FUNCTION "FC21 Ventil 1A0-2E" : VOID	// FC 21
TITLE = Block for valve actuation and fault monitoring
//Erstellung:
//Datum        Bearbeiter                                                 Version
//--------------------------------------------------------------------------------
//26.06.97     H.Rüttling (rh)                                            01.00.00
//
//Änderungen:
//Nr. Datum    Bearb Änderung                                       Marke  Version
//--------------------------------------------------------------------------------
//01  09.02.99 sra   Einfügen der Handbedienuung                    ()    01.01.00
//02  16.04.99 sra   Fehlerbeseitigung Störungsquittierung          ()    01.01.01
//03  21.05.99 jm    Ventiltyp 0 eingefügt                          ()    01.02.00
//04  23.07.99 sra   Ausg. wird auch bei Simulation gesetzt         ()    01.02.01
//06  18.09.00 sra   komplette Überarbeitung / neue Struktur        ()    02.00.00
//07  31.10.05 sra   Ansteuerung Handbedienung im Automode rücksetz.
//                   Handbedienung zentral sperren                  (007) 02.01.00
//08  04.09.06 sra   Änderung Störungsquittierung                   (008) 02.02.00
//09  18.02.09 kmj   Objektststatus für OP ergänzt                  (009) 02.03.00
//10  20.03.09 kal   Objektststatus für OP ergänzt (überarbeitet)   (010) 02.03.01
//11  25.03.09 kal   1A0E-Objekt kann verzögert "in Betrieb" melden (011) 02.03.02
//12  25.03.09 kal   INC nach + geändert                            (012) 02.03.03
//13  20.11.07 gea   Handmode zurücksetzen wenn Handmode gesperrt   (013) 02.03.04
//14  14.07.09 kal   Objektstatus überarbeitet                      (014) 02.03.05
//15  05.12.13 sra   "Anlage ein" eingefügt (Not-Aus-Konzept)       (015) 02.04.00
//________________________________________________________________________________
//Funktion:
//
//-Der Parameter VENTIL_TYP unterscheidet zwischen 4 verschiedenen Ventiltypen
// Typ 0 = Ventil ohne Rückmeldung
// Typ 1 = Ventil oder Klappe mit der Rückmeldung angesteuert und nicht 
//        angesteuert: 1. Ausgang auf, Eingang auf, Eingang zu
//                     2. Ausgang zu , Eingang zu , Eingang auf
// TYP 2 = Ventil oder Klappe mit der Rückmeldung angesteuert
//                     1. Ausgang auf, Eingang auf
//                     2. Ausgang zu , Eingang zu 
// TYP 3 = Ventil oder Klappe mit der Rückmeldung nicht angesteuert
//                     1. Ausgang auf, Eingang zu
//                     2. Ausgang zu , Eingang auf 
//
//-Der Baustein steuert den Ablauf eines Ventils mit 1 Ausgang und 0-2 Eingängen
// durch setzten des Eingangsparameters "in_Ansteuerung_Ventil".
//
//-Der Ausgang wird nur angesteuert wenn der Eingang "in_Anlage_ein" = true
// ist. Diese Funktion ist vorhanden, um bei einem Not-Halt die Anlage vor 
// unkontrolliertem Einschalten zu schützen. 
//
//-Ist in der Ventilstruktur die Taktfunktion freigegeben wird bei Freigabe des 
// Ventils der Ausgang entsprechend der Impuls-/Pausezeit angesteuert.
//
//-Der Baustein überwacht den Zustand des Ausgangs und der Eingänge und generiert 
// nach Ablauf der "Sollzeit Störung" eine Störmeldung
//
//-Ist das Bit "Simulation" auf TRUE, so werden die Eingänge simuliert.
//
//-Ist die Kennung "Schalthäufigkeitszähler_ein" aktiviert werden die
// Ansteuerungen des Ventils aufsummiert. Dies erfolgt mit setzen des Ausgangs.
//
//-Der Baustein kopiert die Parameter "in_Eingang_...", "io_Ausgang_Ventil", 
// "in_Quitt_Stoerung" und "io_Stoerung" in die angegebene Datenstruktur zur 
// Visualisierung auf einem Farbgrafiksystem. Diese Parameter müssen folglich 
// nicht mehr extern umkopiert werden.
//
//-Ist der Parameter "in_Handbedienung_erlaubt" angewählt kann das Ventil über 
// eine Farbgrafik oder ein Bedienterminal manuell angesteuert werden
//
AUTHOR : rh
FAMILY : AZO
VERSION : 0.0
VAR_INPUT
  in_Ventil_Typ : INT ;	//see Functional description below
  in_Handbedienung_erlaubt : BOOL ;	//1 = manual operation permitted, 0 = manual operation not permitted/locked
  in_Quitt_Stoerung_noetig : BOOL ;	//1 = fault acknowledgement required, 0 = automatic fault acknowledgement
  in_Quitt_Stoerung : BOOL ;	//Fault acknowledgement when fault_acknowledgement_required = 1
  in_Anlage_ein : BOOL ;	//Anlage bzw. Anlagenbereich nach Not-Halt freigegeben
  in_Ansteuerung_Ventil : BOOL ;	//Actuation of valve in automatic mode
  in_Eingang_angesteuert : BOOL ;	//Valve intake when actuated
  in_Eingang_nicht_angest : BOOL ;	//Valve intake when not actuated
END_VAR
VAR_IN_OUT
  io_Ausgang_Ventil : BOOL ;	//Valve outlet
  io_Ventil_in_Betrieb : BOOL ;	//Signal "valve in operation" (actuated)
  io_Stoerung : BOOL ;	//Signal "valve fault"
  io_Ventilstruktur : ANY ;	//ANY pointer of valve structure
END_VAR
VAR_TEMP
  Freigabe_Takt : BOOL ;
  Rueckmeldung : BOOL ;
  Start_mit_Impuls : BOOL ;
  Dauertakt : BOOL ;
  Taktausgang : BOOL ;
  Taktanzahl_erreicht : BOOL ;
  Diskrepanz : BOOL ;
  positive_Flanke : BOOL ;
  Impulszeit : REAL ;
  Pausezeit : REAL ;
  Sollanzahl_Takte : INT ;
  Zeitzaehler : REAL ;
  Taktzaehler : INT ;
  Objektstatus : INT ;
END_VAR
BEGIN
NETWORK
TITLE = Anfangs-DW der Struktur aus ANY-Zeiger auslesen
      L     P##io_Ventilstruktur;
      LAR2;
      L     D [AR2,P#6.0];
      LAR2;
NETWORK
TITLE = Simulation
      AN    DIX [AR2,P#3.5];	// Simulation ein (Struktur)
      JC    ESIM;
      A     #io_Ausgang_Ventil;
      =     #in_Eingang_angesteuert;
      AN    #io_Ausgang_Ventil;
      =     #in_Eingang_nicht_angest;
      L     #in_Ventil_Typ;
      L     3;
      <>I;
      JC    ESIM;
      CLR;
      =     #in_Eingang_angesteuert;
      AN    #io_Ausgang_Ventil;
      =     #in_Eingang_nicht_angest;
ESIM: NOP   0;
NETWORK
TITLE = Umschaltung Hand-/Automatikmode 
      A     DIX [AR2,P#2.7];	// Handmode von Farbgrafik (Struktur)
      AN    DIX [AR2,P#3.1];	// Handmode gesperrt (Struktur)
      AN    "M0.0 LockManualMode";	// Handbedienung zentral sperren (007)
      S     DIX [AR2,P#2.6];	// Handmode zu Farbgrafik (Struktur)
      ON    DIX [AR2,P#2.7];	// Handmode von Farbgrafik (Struktur)
      ON    #in_Handbedienung_erlaubt;
      O     "M0.0 LockManualMode";	// Handbedienung zentral sperren (007)
      O     DIX [AR2,P#3.1];	// Handmode gesperrt (Struktur)//(013)
      R     DIX [AR2,P#2.6];	// Handmode zu Farbgrafik (Struktur)
      R     DIX [AR2,P#2.7];	// Handmode von Farbgrafik (Struktur) (007)
NETWORK
TITLE = Ansteuerung Handmode zurücksetzen
//(007) 
      AN    DIX [AR2,P#2.6];	// Handmode zu Farbgrafik (Struktur)
      R     DIX [AR2,P#3.0];	// Ansteuerung Handmode von Farbgrafik (Struktur)
NETWORK
TITLE = Daten für Takt in temporäre Variablen laden
      A     #in_Anlage_ein;	// (015)
      A     #in_Ansteuerung_Ventil;
      A     DIX [AR2,P#3.6];	// Freigabe Takt (Struktur)
      =     #Freigabe_Takt;
      A     DIX [AR2,P#3.2];	// Start mit Impuls (Struktur)
      =     #Start_mit_Impuls;
      A     DIX [AR2,P#3.3];	// Taktanzahl erreicht (Struktur)
      =     #Taktanzahl_erreicht;
      A     DIX [AR2,P#3.4];	// Dauertakt (Struktur)
      =     #Dauertakt;
      A     DIX [AR2,P#3.7];	// Taktausgang (Struktur)
      =     #Taktausgang;
      L     DID [AR2,P#8.0];	// Impulszeit (Struktur)
      T     #Impulszeit;
      L     DID [AR2,P#12.0];	// Pausezeit (Struktur)
      T     #Pausezeit;
      L     DID [AR2,P#16.0];	// Impuls-/Pausezähler (Struktur)
      T     #Zeitzaehler;
      L     DIW [AR2,P#20.0];	// Sollanzahl Takte (Struktur)
      T     #Sollanzahl_Takte;
      L     DIW [AR2,P#22.0];	// Taktzähler (Struktur)
      T     #Taktzaehler;
NETWORK
TITLE = Rückmeldung für Takt
      A(;
      L     #in_Ventil_Typ;
      L     0;
      ==I;
      );
      A     #io_Ausgang_Ventil;
      O;
      A(;
      L     #in_Ventil_Typ;
      L     1;
      ==I;
      );
      A     #in_Eingang_angesteuert;
      O;
      A(;
      L     #in_Ventil_Typ;
      L     2;
      ==I;
      );
      A     #in_Eingang_angesteuert;
      O;
      A(;
      L     #in_Ventil_Typ;
      L     3;
      ==I;
      );
      AN    #in_Eingang_nicht_angest;
      =     #Rueckmeldung;
NETWORK
TITLE = Takt generieren
      CALL  "FC2 Taktgeber_Timernachb" (
           in_Freigabe              := #Freigabe_Takt,
           in_Rueckmeldung          := #Rueckmeldung,
           in_Start_mit_Impuls      := #Start_mit_Impuls,
           in_Dauertakt             := #Dauertakt,
           in_Impuls                := "M1.7 ClockTimerFunction",
           in_Impulszeit_in_100ms   := "MW 6 Timer Val Cycle FCs",
           in_Impulszeit            := #Impulszeit,
           in_Pausezeit             := #Pausezeit,
           in_Sollanzahl_Takte      := #Sollanzahl_Takte,
           io_Taktausgang           := #Taktausgang,
           io_Taktanzahl_erreicht   := #Taktanzahl_erreicht,
           io_Zeitzaehler           := #Zeitzaehler,
           io_Taktzaehler           := #Taktzaehler);
NETWORK
TITLE = Ansteuerung Ventil
      A     #in_Anlage_ein;	// (015)
      A(;
      ON    #in_Quitt_Stoerung_noetig;
      O;
      A     #in_Quitt_Stoerung_noetig;
      AN    #io_Stoerung;
      );
      A(;
      AN    DIX [AR2,P#2.6];	// Automatikmode zu Farbgrafik (Struktur)
      AN    DIX [AR2,P#3.6];	// Freigabe Takt (Struktur)
      A     #in_Ansteuerung_Ventil;
      O;
      AN    DIX [AR2,P#2.6];	// Automatikmode zu Farbgrafik (Struktur)
      A     DIX [AR2,P#3.6];	// Freigabe Takt (Struktur)
      A     #Taktausgang;
      O;
      A     DIX [AR2,P#2.6];	// Handmode zu Farbgrafik (Struktur)
      A     DIX [AR2,P#3.0];	// Ansteuerung Handmode von Farbgrafik (Struktur)
      );
      =     #io_Ausgang_Ventil;
NETWORK
TITLE = Ventiltyp festlegen
      L     #in_Ventil_Typ;
      L     0;
      ==I;
      JC    TYP0;	// Sprung zu Ventil Typ 0
      TAK;
      L     1;
      ==I;
      JC    TYP1;	// Sprung zu Ventil Typ 1
      TAK;
      L     2;
      ==I;
      JC    TYP2;	// Sprung zu Ventil Typ 2
      TAK;
      L     3;
      ==I;
      JC    TYP3;	// Sprung zu Ventil Typ 3
      JU    ENDE;
NETWORK
TITLE = Betriebsmeldung Typ 0 (kein Eingang)
TYP0: A     #io_Ausgang_Ventil;
      A(;	// (011)
      L     DIW [AR2,P#40.0];	// (011) Istzeit Verzögerung (Struktur) 
      L     DIW [AR2,P#38.0];	// (011) Sollzeit Verzögerung (Struktur)
      >=I;	// (011)
      );	// (011)
      =     #io_Ventil_in_Betrieb;	// Betriebsmeldung anzeigen
NETWORK
TITLE = Istzähler Verzögerung hochzählen (011)
      A     #io_Ausgang_Ventil;
      AN    "M4.5 ImpulseClock1,0Sec";	// Sekundenimpuls (Standardmerker)
      O     #io_Ventil_in_Betrieb;	// Betriebsmeldung anzeigen
      JC    KVZ;
      L     DIW [AR2,P#40.0];	// Istzeit Verzögerung (Struktur)
      +     1;
      T     DIW [AR2,P#40.0];	// Istzeit Verzögerung (Struktur)
KVZ:  NOP   0;
NETWORK
TITLE = Istzähler Verzögerung zurücksetzen (011)
      O     #io_Ausgang_Ventil;
      JC    RVZ;
      L     0;
      T     DIW [AR2,P#40.0];	// Istzeit Verzögerung (Struktur)
RVZ:  NOP   0;
NETWORK
TITLE = Diskrepanz Typ 0 (kein Eingang)
      CLR;	// keine Diskrepanz möglich
      =     #Diskrepanz;
      JU    STOE;
NETWORK
TITLE = Betriebsmeldung Typ1 (Eingang angesteuert und nicht angesteuert)
TYP1: A     #io_Ausgang_Ventil;
      A     #in_Eingang_angesteuert;
      AN    #in_Eingang_nicht_angest;
      =     #io_Ventil_in_Betrieb;
NETWORK
TITLE = Diskrepanz Typ 1 (Eingang angesteuert und nicht angesteuert)
      A     #io_Ausgang_Ventil;
      AN    #in_Eingang_angesteuert;
      O;
      AN    #io_Ausgang_Ventil;
      AN    #in_Eingang_nicht_angest;
      O;
      A     #in_Eingang_angesteuert;
      A     #in_Eingang_nicht_angest;
      O;
      AN    #in_Eingang_angesteuert;
      AN    #in_Eingang_nicht_angest;
      =     #Diskrepanz;
      JU    STOE;
NETWORK
TITLE = Betriebsmeldung Typ 2 (Eingang angesteuert)
TYP2: A     #io_Ausgang_Ventil;
      A     #in_Eingang_angesteuert;
      =     #io_Ventil_in_Betrieb;
NETWORK
TITLE = Diskrepanz Typ 2 (Eingang angesteuert)
      A     #io_Ausgang_Ventil;
      AN    #in_Eingang_angesteuert;
      O;
      AN    #io_Ausgang_Ventil;
      A     #in_Eingang_angesteuert;
      =     #Diskrepanz;
      JU    STOE;
NETWORK
TITLE = Betriebsmeldung Typ 3 (Eingang nicht angesteuert)
TYP3: A     #io_Ausgang_Ventil;
      AN    #in_Eingang_nicht_angest;
      =     #io_Ventil_in_Betrieb;
NETWORK
TITLE = Diskrepanz Typ 3 (Eingang nicht angesteuert)
      A     #io_Ausgang_Ventil;
      A     #in_Eingang_nicht_angest;
      O;
      AN    #io_Ausgang_Ventil;
      AN    #in_Eingang_nicht_angest;
      =     #Diskrepanz;
NETWORK
TITLE = Störungszähler
STOE: A     #in_Quitt_Stoerung_noetig;
      AN    #in_Quitt_Stoerung;
      A     #io_Stoerung;
      O;
      A     #Diskrepanz;
      AN    #in_Quitt_Stoerung;	// (008)
      O;	// (008)
      AN    #in_Quitt_Stoerung_noetig;	// (008)
      A     #Diskrepanz;	// (008)
      JC    SZ1;
      L     0;	// Wenn keine Diskrepanz dann Zähler löschen
      T     DIW [AR2,P#6.0];	// Istzeit Störung (Struktur)
      JU    ESZ;
// Störungszähler in jeder Sekunde erhöhen
SZ1:  O     #io_Stoerung;
      ON    "M4.5 ImpulseClock1,0Sec";	// Sekundenimpuls (Standardmerker)
      JC    ESZ;
      L     DIW [AR2,P#6.0];	// Istzeit Störung (Struktur)
      +     1;	// (012)
      T     DIW [AR2,P#6.0];	// Istzeit Störung (Struktur)
ESZ:  NOP   0;
NETWORK
TITLE = Störmeldung ausgeben
      L     DIW [AR2,P#6.0];	// Istzeit Störung (Struktur)
      L     DIW [AR2,P#4.0];	// Sollzeit Störung (Struktur)
      >=I;
      =     #io_Stoerung;
NETWORK
TITLE = Stoerung quittieren
      O     #Diskrepanz;	// Stoerung steht noch an
      ON    #io_Stoerung;
      JC    ESQ;
      ON    #in_Quitt_Stoerung_noetig;	// Stoerung muß quittiert werden ?
      JC    SQ1;	// Stoerung muß nicht quittiert werden
      A     #in_Quitt_Stoerung;
SQ1:  R     #io_Stoerung;
ESQ:  NOP   0;
NETWORK
TITLE = Flankenauswertung Ausgang Ventil für Schalthäufigkeitzähler
      A     #io_Ausgang_Ventil;
      FP    DIX [AR2,P#24.3];	// Flankenmerker Ausgang (Struktur)
      =     #positive_Flanke;
NETWORK
TITLE = Schalthäufigkeitzähler
      ON    DIX [AR2,P#0.3];	// Kennung Schalthäufigkeitzähler ein (Struktur)
      ON    #positive_Flanke;
      JC    ESHZ;
      L     1.000000e+00;
      L     DID [AR2,P#26.0];	// Schalthäufigkeitzähler (Struktur)
      +R;
      T     DID [AR2,P#26.0];	// Schalthäufigkeitzähler (Struktur)
ESHZ: NOP   0;
NETWORK
TITLE = Schalthäufigkeitzähler zurücksetzten
      AN    DIX [AR2,P#24.0];	// Reset Schalthäufigkeitzähler (Struktur)
      JC    E_RS;
      L     0.000000e+00;
      T     DID [AR2,P#26.0];	// Schalthäufigkeitzähler (Struktur)
      CLR;
      =     DIX [AR2,P#24.0];	// Reset Schalthäufigkeitzähler (Struktur)
E_RS: NOP   0;
NETWORK
TITLE = Warnmeldung Schalthäufigkeitszähler erzeugen
      A(;
      L     DID [AR2,P#26.0];	// Schalthäufigkeitzähler (Struktur)
      L     DID [AR2,P#30.0];	// Sollwert Warnung (Struktur)
      >R;
      );
      A(;
      L     DID [AR2,P#30.0];	// Sollwert Warnung (Struktur)
      L     0.000000e+00;
      <>R;
      );
      =     DIX [AR2,P#24.1];	// Warnmeldung Schalthäufigkeitzähler (Struktur)
NETWORK
TITLE = Alarmmeldung Schalthäufigkeitszähler erzeugen
      A(;
      L     DID [AR2,P#26.0];	// Schalthäufigkeitzähler (Struktur)
      L     DID [AR2,P#34.0];	// Sollwert Alarm (Struktur)
      >R;
      );
      A(;
      L     DID [AR2,P#34.0];	// Sollwert Alarm (Struktur)
      L     0.000000e+00;
      <>R;
      );
      =     DIX [AR2,P#24.2];	// Alarmmeldung Schalthäufigkeitzähler (Struktur)
NETWORK
TITLE =  Objektstatus für Visualisation OP (009) (010)
//Stati:
//-------
//1 = nicht in Betrieb, keine Störung ==> Farbvorschlag weiß
//5 = angesteuert, in Betrieb, keine Störung ==> Farbvorschlag grün
//9 = angesteuert, nicht in Betrieb, keine Störung ==> Farbvorschlag grau
//16 = Störung ==> Farbvorschlag rot
// 1 = nicht in Betrieb, keine Störung ==> Farbvorschlag weiß
      L     1;
      AN    #io_Ausgang_Ventil;
      AN    #io_Stoerung;
      AN    DIX [AR2,P#1.3];	// (014) Kennung "invers"
      O;
      A     #io_Ausgang_Ventil;
      A     #io_Ventil_in_Betrieb;
      AN    #io_Stoerung;
      A     DIX [AR2,P#1.3];	// (014) Kennung "invers"
      JC    disp;
// 5 = angesteuert, in Betrieb, keine Störung ==> Farbvorschlag grün
      L     5;
      A     #io_Ausgang_Ventil;
      A     #io_Ventil_in_Betrieb;
      AN    #io_Stoerung;
      AN    DIX [AR2,P#1.3];	// (014) Kennung "invers"
      O;
      AN    #io_Ausgang_Ventil;
      AN    #io_Stoerung;
      A     DIX [AR2,P#1.3];	// (014) Kennung "invers"
      JC    disp;
// 9 = angesteuert, nicht in Betrieb, keine Störung ==> Farbvorschlag grau
      L     9;
      A     #io_Ausgang_Ventil;
      AN    #io_Ventil_in_Betrieb;
      AN    #io_Stoerung;
      JC    disp;
// 16 = Störung ==> Farbvorschlag rot
      L     16;
      A     #io_Stoerung;
      JC    disp;
      L     0;
disp: T     #Objektstatus;
NETWORK
TITLE = Daten in Struktur speichern
      A     #in_Anlage_ein;	// (015)
      =     DIX [AR2,P#42.0];	// (015) Anlage ein (Struktur)
      A     #in_Eingang_angesteuert;
      =     DIX [AR2,P#2.1];	// Eingang angesteuert (Struktur)
      A     #in_Eingang_nicht_angest;
      =     DIX [AR2,P#2.2];	// Eingang nicht angesteuert (Struktur)
      A     #io_Ausgang_Ventil;
      =     DIX [AR2,P#2.0];	// Ausgang Ventil (Struktur)
      A     #io_Ventil_in_Betrieb;
      =     DIX [AR2,P#2.4];	// Ventil in Betrieb (Struktur)
      A     #io_Stoerung;
      =     DIX [AR2,P#2.5];	// Störung (Struktur)
      A     #Taktanzahl_erreicht;
      =     DIX [AR2,P#3.3];	// Taktanzahl erreicht (Struktur)
      A     #Taktausgang;
      =     DIX [AR2,P#3.7];	// Taktausgang (Struktur)
      L     #Zeitzaehler;
      T     DID [AR2,P#16.0];	// Impuls-/Pausezähler (Struktur)
      L     #Taktzaehler;
      T     DIW [AR2,P#22.0];	// Taktzähler (Struktur)
      L     #Objektstatus;	// (009)
      T     DIW [AR2,P#48.0];	// #Objektstatus  (Struktur)   // (009)
NETWORK
TITLE = ENDE
ENDE: NOP   0;
END_FUNCTION

FUNCTION "FC22 Ventil 2A2E" : VOID	// FC 22
TITLE = Block for valve actuation and fault monitoring 2O,2I
//Erstellung:
//Datum        Bearbeiter                                                 Version
//--------------------------------------------------------------------------------
//24.09.98     A.Geiger (gea)                                             01.00.00
//
//Änderungen:
//Nr. Datum    Bearb Änderung                                       Marke  Version
//--------------------------------------------------------------------------------
//01  16.04.99 sra   Fehlerbeseitigung Störungsquittierung          ()    01.00.01
//02  21.05.99 sra   Einfügen der Handbedienuung                    ()    01.01.00
//03  23.07.99 sra   Ausg. wird auch bei Simulation gesetzt         ()    01.01.01
//04  19.10.99 sra   Anpassung an neue Struktur                     ()    01.02.00
//05  19.09.00 sra   komplette Überarbeitung / neue Struktur        ()    02.00.00
//06  15.02.01 sra   Rücksetzen Istwert Störung bei Quitt.          ()    02.00.01
//07  31.03.03 sra   Fehlerbeseitigung Störungsquittierung          (007) 02.00.02
//08  23.03.05 sra   Änderung Störungsquittierung                   (008) 02.01.00
//09  31.10.05 sra   Ansteuerung Handbedienung im Automode rücksetz.
//                   Handbedienung zentral sperren                  (009) 02.02.00
//10  03.05.06 gea   Fehlerbeseitigung Störungszähler               (010) 02.02.01
//11  18.02.09 kmj   Objektstatus ergänzt                           (011) 02.03.00
//12  20.03.09 kal   Objektstatus ergänzt (überarbeitet)            (012) 02.03.01
//13  24.04.09 gea   Handmode zurücksetzen wenn Handmode gesperrt   (013) 02.03.02
//14  10.09.09 sra   Objektststatus für OP ergänzt (erweitert)      (014) 02.04.00
//15  15.10.09 gea   Korrektur Taktpause                            (015) 02.04.01
//16  26.03.12 jm    Objektstatus korrigiert                        (016) 02.04.02
//17  07.09.12 jm    Ohjektstatus aufgeteilt (3 Versionen)          (017) 02.04.03
//18  12.10.12 jm    Objektstatus 3 optimiert                       (018) 02.04.04
//19  15.10.12 jm    Objektstatus 3 optimiert (1,6 anstatt 1,5)     (019) 02.04.05
//20  18.12.12 sra   Kennung links rechts eingefügt                 (020) 02.05.00
//21  05.12.13 sra   "Anlage ein" eingefügt (Not-Aus-Konzept)       (021) 02.06.00
//22  24.07.14 jm    Ohjektstatus ergänzt/geändert                  (022) 02.07.01
//23  09.03.16 jm    Objektstatus 9/19 bis Ende oder Störung        (023) 02.07.02
//________________________________________________________________________________
//Funktion:
//
//-Der Baustein steuert den Ablauf eines Ventils mit 2 Ausgängen und 2 Eingängen.
//
//-Die Ausgänge werden nur angesteuert wenn der Eingang "in_Anlage_ein" = true
// ist. Diese Funktion ist vorhanden, um bei einem Not-Halt die Anlage vor 
// unkontrolliertem Einschalten zu schützen. 
//
//-Ist in der Ventilstruktur die Taktfunktion freigegeben wird bei Freigabe des 
// Ventils der Ausgang entsprechend der Impuls-/Pausezeit angesteuert.
//
//-Der Baustein überwacht den Zustand der Ausgänge und der Eingänge und generiert 
// nach Ablauf der "Sollzeit Störung" eine Störmeldung
//
//-Ist das Bit "Simulation" auf TRUE, so werden die Eingänge simuliert.
//
//-Ist die Kennung "Schalthäufigkeitszähler_ein" aktiviert werden die
// Ansteuerungen des Ventils aufsummiert. Dies erfolgt mit setzen des Ausgangs.
//
//-Der Baustein kopiert die Parameter "in_Eingang_...", "io_Ausgang_...", 
// "in_Quitt_Stoerung" und "io_Stoerung" in die angegebene Datenstruktur zur 
// Visualisierung auf einem Farbgrafiksystem. Diese Parameter müssen folglich 
// nicht mehr extern umkopiert werden.
//
//-Ist der Parameter "in_Handbedienung_erlaubt" angewählt kann das Ventil über 
// eine Farbgrafik oder ein Bedienterminal manuell angesteuert werden
//
AUTHOR : gea
FAMILY : AZO
NAME : standard
VERSION : 0.0
VAR_INPUT
  in_Handbedienung_erlaubt : BOOL ;	//1 = manual operation permitted, 0 = manual operation not permitted/locked
  in_Quitt_Stoerung_noetig : BOOL ;	//1 = fault acknowledgement required, 0 = automatic fault acknowledgement
  in_Quitt_Stoerung : BOOL ;	//Fault acknowledgement when fault_acknowledgement_required = 1
  in_Anlage_ein : BOOL ;	//Anlage bzw. Anlagenbereich nach Not-Halt freigegeben
  in_Ansteuerung_Stellung1 : BOOL ;	//Actuation of valve position 1 in automatic mode
  in_Ansteuerung_Stellung2 : BOOL ;	//Actuation of valve position 2 in automatic mode
  in_Eingang_Stellung_1 : BOOL ;	//Valve intake when position 1 actuated
  in_Eingang_Stellung_2 : BOOL ;	//Valve intake when position 2 actuated
END_VAR
VAR_IN_OUT
  io_Ausgang_Stellung_1 : BOOL ;	//Valve output to actuate position 1
  io_Ausgang_Stellung_2 : BOOL ;	//Valve output to actuate position 2
  io_Stellung_1_Betrieb : BOOL ;	//Signal "position 1 in operation" (position 1 actuated)
  io_Stellung_2_Betrieb : BOOL ;	//Signal "position 2 in operation" (position 2 actuated)
  io_Stoerung : BOOL ;	//Signal "valve fault"
  io_Ventilstruktur : ANY ;	//ANY pointer of valve structure
END_VAR
VAR_TEMP
  Freigabe_Takt : BOOL ;
  Rueckmeldung : BOOL ;
  Start_mit_Impuls : BOOL ;
  Dauertakt : BOOL ;
  Taktausgang : BOOL ;
  Taktanzahl_erreicht : BOOL ;
  Diskrepanz : BOOL ;
  positive_Flanke : BOOL ;
  Impulszeit : REAL ;
  Pausezeit : REAL ;
  Sollanzahl_Takte : INT ;
  Zeitzaehler : REAL ;
  Taktzaehler : INT ;
  Objektstatus : INT ;
END_VAR
BEGIN
NETWORK
TITLE = Anfangs-DW der Struktur aus ANY-Zeiger auslesen
      L     P##io_Ventilstruktur;
      LAR2;
      L     D [AR2,P#6.0];
      LAR2;
NETWORK
TITLE = Simulation
      AN    DIX [AR2,P#4.1];	// Simulation ein (Struktur)
      JC    ESIM;
      A     #io_Ausgang_Stellung_1;
      AN    #io_Ausgang_Stellung_2;
      O;
      AN    #io_Ausgang_Stellung_2;
      AN    DIX [AR2,P#2.2];	// Eingang Stellung 1 (Struktur)
      AN    DIX [AR2,P#2.3];	// Eingang Stellung 2 (Struktur)
      O;
      AN    #io_Ausgang_Stellung_1;
      AN    #io_Ausgang_Stellung_2;
      A     DIX [AR2,P#2.2];	// Eingang Stellung 1 (Struktur)
      S     #in_Eingang_Stellung_1;
      R     #in_Eingang_Stellung_2;
      AN    #io_Ausgang_Stellung_1;
      A     #io_Ausgang_Stellung_2;
      O;
      AN    #io_Ausgang_Stellung_1;
      AN    #io_Ausgang_Stellung_2;
      A     DIX [AR2,P#2.3];	// Eingang Stellung 2 (Struktur)
      R     #in_Eingang_Stellung_1;
      S     #in_Eingang_Stellung_2;
ESIM: NOP   0;
NETWORK
TITLE = Umschaltung Hand-/Automatikmode 
      A     DIX [AR2,P#3.2];	// Handmode von Farbgrafik (Struktur)
      AN    DIX [AR2,P#3.5];	// Handmode gesperrt (Struktur)
      AN    "M0.0 LockManualMode";	// Handbedienung zentral sperren (009)
      S     DIX [AR2,P#3.1];	// Handmode zu Farbgrafik (Struktur)
      ON    DIX [AR2,P#3.2];	// Handmode von Farbgrafik (Struktur)
      ON    #in_Handbedienung_erlaubt;
      O     "M0.0 LockManualMode";	// Handbedienung zentral sperren (009)
      O     DIX [AR2,P#3.5];	// Handmode gesperrt (Struktur) (013)
      R     DIX [AR2,P#3.1];	// Handmode zu Farbgrafik (Struktur)
      R     DIX [AR2,P#3.2];	// Handmode von Farbgrafik (Struktur) (009)
NETWORK
TITLE = Ansteuerung Handmode zurücksetzen
//(009) 
      AN    DIX [AR2,P#3.1];	// Handmode zu Farbgrafik (Struktur)
      R     DIX [AR2,P#3.3];	// Ansteuerung Stellung 1 Handmode von Farbgrafik (Struktur)
      R     DIX [AR2,P#3.4];	// Ansteuerung Stellung 2 Handmode von Farbgrafik (Struktur)
NETWORK
TITLE = Daten für Takt in temporäre Variablen laden
      A     #in_Anlage_ein;	// (021)
      A(;
      O     #in_Ansteuerung_Stellung1;
      O     #in_Ansteuerung_Stellung2;
      );
      A     DIX [AR2,P#4.2];	// Freigabe Takt (Struktur)
      =     #Freigabe_Takt;
      A     DIX [AR2,P#3.6];	// Start mit Impuls (Struktur)
      =     #Start_mit_Impuls;
      A     DIX [AR2,P#3.7];	// Taktanzahl erreicht (Struktur)
      =     #Taktanzahl_erreicht;
      A     DIX [AR2,P#4.0];	// Dauertakt (Struktur)
      =     #Dauertakt;
      A     DIX [AR2,P#4.3];	// Taktausgang (Struktur)
      =     #Taktausgang;
      L     DID [AR2,P#10.0];	// Impulszeit (Struktur)
      T     #Impulszeit;
      L     DID [AR2,P#14.0];	// Pausezeit (Struktur)
      T     #Pausezeit;
      L     DID [AR2,P#18.0];	// Impuls-/Pausezähler (Struktur)
      T     #Zeitzaehler;
      L     DIW [AR2,P#22.0];	// Sollanzahl Takte (Struktur)
      T     #Sollanzahl_Takte;
      L     DIW [AR2,P#24.0];	// Taktzähler (Struktur)
      T     #Taktzaehler;
NETWORK
TITLE = Rückmeldung für Takt
// (network holds code this reader does not know; not shown)
NETWORK
TITLE = Takt generieren
      CALL  "FC2 Taktgeber_Timernachb" (
           in_Freigabe              := #Freigabe_Takt,
           in_Rueckmeldung          := #Rueckmeldung,
           in_Start_mit_Impuls      := #Start_mit_Impuls,
           in_Dauertakt             := #Dauertakt,
           in_Impuls                := "M1.7 ClockTimerFunction",
           in_Impulszeit_in_100ms   := "MW 6 Timer Val Cycle FCs",
           in_Impulszeit            := #Impulszeit,
           in_Pausezeit             := #Pausezeit,
           in_Sollanzahl_Takte      := #Sollanzahl_Takte,
           io_Taktausgang           := #Taktausgang,
           io_Taktanzahl_erreicht   := #Taktanzahl_erreicht,
           io_Zeitzaehler           := #Zeitzaehler,
           io_Taktzaehler           := #Taktzaehler);
NETWORK
TITLE = Ansteuerung Stellung 1
      A     #in_Anlage_ein;	// (021)
      A(;
      ON    #in_Quitt_Stoerung_noetig;
      O;
      A     #in_Quitt_Stoerung_noetig;
      AN    #io_Stoerung;
      );
      A(;
      AN    DIX [AR2,P#3.1];	// Automatikmode zu Farbgrafik (Struktur)
      AN    DIX [AR2,P#4.2];	// Freigabe Takt (Struktur)
      A     #in_Ansteuerung_Stellung1;
      AN    #in_Ansteuerung_Stellung2;
      O;
      AN    DIX [AR2,P#3.1];	// Automatikmode zu Farbgrafik (Struktur)
      A     DIX [AR2,P#4.2];	// Freigabe Takt (Struktur)
      A     #Taktausgang;
      O;
      A     DIX [AR2,P#3.1];	// Handmode zu Farbgrafik (Struktur)
      A     DIX [AR2,P#3.3];	// Ansteuerung Stellung 1 Handmode von Farbgrafik (Struktur)
      AN    DIX [AR2,P#3.4];	// Ansteuerung Stellung 2 Handmode von Farbgrafik (Struktur)
      );
      =     #io_Ausgang_Stellung_1;
NETWORK
TITLE = Ansteuerung Stellung 2
      A     #in_Anlage_ein;	// (021)
      A(;
      ON    #in_Quitt_Stoerung_noetig;
      O;
      A     #in_Quitt_Stoerung_noetig;
      AN    #io_Stoerung;
      );
      A(;
      AN    DIX [AR2,P#3.1];	// Automatikmode zu Farbgrafik (Struktur)
      AN    DIX [AR2,P#4.2];	// Freigabe Takt (Struktur)
      A     #in_Ansteuerung_Stellung2;
      AN    #in_Ansteuerung_Stellung1;
      O;
      AN    DIX [AR2,P#3.1];	// Automatikmode zu Farbgrafik (Struktur)
      A     DIX [AR2,P#4.2];	// Freigabe Takt (Struktur)
      AN    #Taktausgang;
      O;
      A     DIX [AR2,P#3.1];	// Handmode zu Farbgrafik (Struktur)
      AN    DIX [AR2,P#3.3];	// Ansteuerung Stellung 1 Handmode von Farbgrafik (Struktur)
      A     DIX [AR2,P#3.4];	// Ansteuerung Stellung 2 Handmode von Farbgrafik (Struktur)
      );
      =     #io_Ausgang_Stellung_2;
NETWORK
TITLE = Betriebsmeldung Stellung 1
      A     #io_Ausgang_Stellung_1;
      A     #in_Eingang_Stellung_1;
      AN    #io_Ausgang_Stellung_2;
      AN    #in_Eingang_Stellung_2;
      =     #io_Stellung_1_Betrieb;
NETWORK
TITLE = Betriebsmeldung Stellung 2
      AN    #io_Ausgang_Stellung_1;
      AN    #in_Eingang_Stellung_1;
      A     #io_Ausgang_Stellung_2;
      A     #in_Eingang_Stellung_2;
      =     #io_Stellung_2_Betrieb;
NETWORK
TITLE = Diskrepanz
      A     #io_Ausgang_Stellung_1;	// Nicht auf Abzweig
      AN    #in_Eingang_Stellung_1;
      O;
      A     #io_Ausgang_Stellung_2;	// Nicht auf Gerade
      AN    #in_Eingang_Stellung_2;
      O;
      A     #in_Eingang_Stellung_1;	// Stellung nicht definiert
      A     #in_Eingang_Stellung_2;
      O;
      AN    #in_Eingang_Stellung_1;	// Stellung nicht definiert
      AN    #in_Eingang_Stellung_2;
      O;
      A     #in_Ansteuerung_Stellung1;	// Ansteuerung nicht zulässig
      A     #in_Ansteuerung_Stellung2;
      =     #Diskrepanz;	// Diskrepanz feststellen
NETWORK
TITLE = Störungszähler
      A     #in_Quitt_Stoerung_noetig;
      AN    #in_Quitt_Stoerung;
//      U     #Diskrepanz                 // (007)
      A     #io_Stoerung;
      O;
//      UN    #in_Quitt_Stoerung_noetig   // (007)
      A     #Diskrepanz;
      AN    #in_Quitt_Stoerung;	// (008)
      O;	// (010)
      AN    #in_Quitt_Stoerung_noetig;	// (010)
      A     #Diskrepanz;	// (010)
      JC    SZ1;
      L     0;	// Wenn keine Diskrepanz dann Zähler löschen
      T     DIW [AR2,P#8.0];	// Istzeit Störung (Struktur)
      JU    ESZ;
// Störungszähler in jeder Sekunde erhöhen
SZ1:  O     #io_Stoerung;
      ON    "M4.5 ImpulseClock1,0Sec";	// Sekundenimpuls (Standardmerker)
      JC    ESZ;
      L     DIW [AR2,P#8.0];	// Istzeit Störung (Struktur)
      INC   1;
      T     DIW [AR2,P#8.0];	// Istzeit Störung (Struktur)
ESZ:  NOP   0;
NETWORK
TITLE = Störmeldung ausgeben
      L     DIW [AR2,P#8.0];	// Istzeit Störung (Struktur)
      L     DIW [AR2,P#6.0];	// Sollzeit Störung (Struktur)
      >=I;
      =     #io_Stoerung;
NETWORK
TITLE = Stoerung quittieren
      O     #Diskrepanz;	// Stoerung steht noch an
      ON    #io_Stoerung;
      JC    ESQ;
      ON    #in_Quitt_Stoerung_noetig;	// Stoerung muß quittiert werden ?
      JC    SQ1;	// Stoerung muß nicht quittiert werden
      A     #in_Quitt_Stoerung;
SQ1:  R     #io_Stoerung;
ESQ:  NOP   0;
NETWORK
TITLE = Flankenauswertung Ausgang Ventil für Schalthäufigkeitzähler
//Es wird die Schalthäufigkeit der Ventile gezählt !  
      A     #io_Ausgang_Stellung_1;
      A     #in_Eingang_Stellung_1;
      O;
      A     #io_Ausgang_Stellung_2;
      A     #in_Eingang_Stellung_2;
      FP    DIX [AR2,P#26.3];	// Flankenmerker Ausgang (Struktur)
      =     #positive_Flanke;
NETWORK
TITLE = Schalthäufigkeitzähler
      ON    DIX [AR2,P#0.3];	// Kennung Schalthäufigkeitzähler ein (Struktur)
      ON    #positive_Flanke;
      JC    ESHZ;
      L     1.000000e+00;
      L     DID [AR2,P#28.0];	// Schalthäufigkeitzähler (Struktur)
      +R;
      T     DID [AR2,P#28.0];	// Schalthäufigkeitzähler (Struktur)
ESHZ: NOP   0;
NETWORK
TITLE = Schalthäufigkeitzähler zurücksetzten
      AN    DIX [AR2,P#26.0];	// Reset Schalthäufigkeitzähler (Struktur)
      JC    E_RS;
      L     0.000000e+00;
      T     DID [AR2,P#28.0];	// Schalthäufigkeitzähler (Struktur)
      CLR;
      =     DIX [AR2,P#26.0];	// Reset Schalthäufigkeitzähler (Struktur)
E_RS: NOP   0;
NETWORK
TITLE = Warnmeldung Schalthäufigkeitzähler erzeugen
      A(;
      L     DID [AR2,P#28.0];	// Schalthäufigkeitzähler (Struktur)
      L     DID [AR2,P#32.0];	// Sollwert Warnung (Struktur)
      >R;
      );
      A(;
      L     DID [AR2,P#32.0];	// Sollwert Warnung (Struktur)
      L     0.000000e+00;
      <>R;
      );
      =     DIX [AR2,P#26.1];	// Warnmeldung Schalthäufigkeitzähler (Struktur)
NETWORK
TITLE = Alarmmeldung Schalthäufigkeitzähler erzeugen
      A(;
      L     DID [AR2,P#28.0];	// Schalthäufigkeitzähler (Struktur)
      L     DID [AR2,P#36.0];	// Sollwert Alarm (Struktur)
      >R;
      );
      A(;
      L     DID [AR2,P#36.0];	// Sollwert Alarm (Struktur)
      L     0.000000e+00;
      <>R;
      );
      =     DIX [AR2,P#26.2];	// Alarmmeldung Schalthäufigkeitzähler (Struktur)
NETWORK
TITLE = Objektstatus für Visualisation OP (011)(012)(017)
//Stati:
//-------
//1 = nicht angesteuert, Ventil in Position 1, keine Störung ==> grau
//2 = nicht angesteuert, Ventil in Position 2, keine Störung ==> grau
//5 = Position 1 angesteuert, Ventil in Position 1, keine Störung ==> grün
//6 = Position 2 angesteuert, Ventil in Position 2, keine Störung ==> grün
//9 = Position 1 angesteuert, Ventil nicht in Position 1, keine Störung ==> weiß
//10 = Position 2 angesteuert, Ventil nicht in Position 2, keine Störung ==> weiß
//14 = Störung, quittierpflichtig, Ausgang nicht angesteuert, Störung ==> rot/weiß
//15 = Störung, nicht quittierpflichtig, Ausgang angesteuert, Störung ==> rot/grün
//16 = Störung quittiert ==> rot
      A(;
      O     DIX [AR2,P#0.7];	// Kennung "gerade/abzweig"
      O     DIX [AR2,P#1.0];	// Kennung "Stellung1/Stellung2"
      O     DIX [AR2,P#1.6];	// Kennung "links/rechts"               (020)
      );
      JCN   NSV1;	// Not Status Version 1
// 1 ==> grau
      L     1;
      AN    #io_Stoerung;
      A(;
      AN    DIX [AR2,P#0.5];	// Kennung "invers"
      A     #in_Eingang_Stellung_1;
      AN    #in_Eingang_Stellung_2;
      AN    #io_Ausgang_Stellung_1;
      AN    #io_Ausgang_Stellung_2;
      O;
      A     DIX [AR2,P#0.5];	// Kennung "invers"
      AN    #in_Eingang_Stellung_1;
      A     #in_Eingang_Stellung_2;
      AN    #io_Ausgang_Stellung_1;
      AN    #io_Ausgang_Stellung_2;
      );
      JC    disp;
// 2 ==> grau
      L     2;
      AN    #io_Stoerung;
      A(;
      AN    DIX [AR2,P#0.5];	// Kennung "invers"
      AN    #in_Eingang_Stellung_1;
      A     #in_Eingang_Stellung_2;
      AN    #io_Ausgang_Stellung_1;
      AN    #io_Ausgang_Stellung_2;
      O;
      A     DIX [AR2,P#0.5];	// Kennung "invers"
      A     #in_Eingang_Stellung_1;
      AN    #in_Eingang_Stellung_2;
      AN    #io_Ausgang_Stellung_1;
      AN    #io_Ausgang_Stellung_2;
      );
      JC    disp;
// 5 ==> grün
      L     5;
      AN    #io_Stoerung;
      A(;
      AN    DIX [AR2,P#0.5];	// Kennung "invers"
      A     #in_Eingang_Stellung_1;
      AN    #in_Eingang_Stellung_2;
      A     #io_Ausgang_Stellung_1;
      AN    #io_Ausgang_Stellung_2;
      O;
      A     DIX [AR2,P#0.5];	// Kennung "invers"
      AN    #in_Eingang_Stellung_1;
      A     #in_Eingang_Stellung_2;
      AN    #io_Ausgang_Stellung_1;
      A     #io_Ausgang_Stellung_2;
      );
      JC    disp;
// 6 ==> grün
      L     6;
      AN    #io_Stoerung;
      A(;
      AN    DIX [AR2,P#0.5];	// Kennung "invers"
      AN    #in_Eingang_Stellung_1;
      A     #in_Eingang_Stellung_2;
      AN    #io_Ausgang_Stellung_1;
      A     #io_Ausgang_Stellung_2;
      O;
      A     DIX [AR2,P#0.5];	// Kennung "invers"
      A     #in_Eingang_Stellung_1;
      AN    #in_Eingang_Stellung_2;
      A     #io_Ausgang_Stellung_1;
      AN    #io_Ausgang_Stellung_2;
      );
      JC    disp;
// 9 ==> weiß
      L     9;
      AN    #io_Stoerung;
      A(;
      AN    DIX [AR2,P#0.5];	// Kennung "invers"
      AN    #in_Eingang_Stellung_1;
//      UN    #in_Eingang_Stellung_2    // (023)
      A     #io_Ausgang_Stellung_1;
      AN    #io_Ausgang_Stellung_2;
      O;
      A     DIX [AR2,P#0.5];	// Kennung "invers"
//      UN    #in_Eingang_Stellung_1    // (023)
      AN    #in_Eingang_Stellung_2;
      AN    #io_Ausgang_Stellung_1;
      A     #io_Ausgang_Stellung_2;
      );
      JC    disp;
// 10 ==> weiß
      L     10;
      AN    #io_Stoerung;
      A(;
      AN    DIX [AR2,P#0.5];	// Kennung "invers"
//      UN    #in_Eingang_Stellung_1    // (023)
      AN    #in_Eingang_Stellung_2;
      AN    #io_Ausgang_Stellung_1;
      A     #io_Ausgang_Stellung_2;
      O;
      A     DIX [AR2,P#0.5];	// Kennung "invers"
      AN    #in_Eingang_Stellung_1;
//      UN    #in_Eingang_Stellung_2    // (023)
      A     #io_Ausgang_Stellung_1;
      AN    #io_Ausgang_Stellung_2;
      );
      JC    disp;
// 14 = Störung, quittierpflichtig, Ausgang nicht angesteuert, Störung ==> rot/weiß
      L     14;	// (014)
      A     #io_Stoerung;	// (014)
      AN    #in_Quitt_Stoerung;	// (014)
      AN    #io_Ausgang_Stellung_1;	// (014)
      AN    #io_Ausgang_Stellung_2;	// (014)
      JC    disp;	// (014)
// 15 = Störung, nicht quittierpflichtig, Ausgang angesteuert, Störung ==> rot/grün
      L     15;	// (014)
      A     #io_Stoerung;	// (014)
      AN    #in_Quitt_Stoerung;	// (014)
      A(;	// (014)
      O     #io_Ausgang_Stellung_1;	// (014)
      O     #io_Ausgang_Stellung_2;	// (014)
      );	// (014)
      JC    disp;	// (014)
// 16 = Störung quittiert ==> rot
      L     16;
      A     #io_Stoerung;
      JC    disp;
NSV1: NOP   0;
NETWORK
TITLE = Objektstatus für Visualisation OP (011)(012)(017)
//Stati:
//-------
//1 = nicht angesteuert, Ventil in Position 1, keine Störung ==> grau
//2 = nicht angesteuert, Ventil in Position 2, keine Störung ==> grau
//5 = Position 1 angesteuert, Ventil in Position 1, keine Störung ==> grün
//6 = Position 2 angesteuert, Ventil in Position 2, keine Störung ==> grün
//9 = Position 1 angesteuert, Ventil nicht in Position 1, keine Störung ==> weiß
//10 = Position 2 angesteuert, Ventil nicht in Position 2, keine Störung ==> weiß
//14 = Störung, quittierpflichtig, Ausgang nicht angesteuert, Störung ==> rot/weiß
//15 = Störung, nicht quittierpflichtig, Ausgang angesteuert, Störung ==> rot/grün
//16 = Störung quittiert ==> rot
      A(;
//      O     DIX [AR2,P#1.1]             // Kennung "oben/unten" // (022)
      O     DIX [AR2,P#1.2];	// Kennung "grob/fein"
      );
      JCN   NSV2;	// Not Status Version 2
// 1 ==> grau
      L     1;
      AN    #io_Stoerung;
      A(;
      AN    DIX [AR2,P#0.5];	// Kennung "invers"
      AN    #in_Eingang_Stellung_1;
      A     #in_Eingang_Stellung_2;
      AN    #io_Ausgang_Stellung_1;
      AN    #io_Ausgang_Stellung_2;
      O;
      A     DIX [AR2,P#0.5];	// Kennung "invers"
      A     #in_Eingang_Stellung_1;
      AN    #in_Eingang_Stellung_2;
      AN    #io_Ausgang_Stellung_1;
      AN    #io_Ausgang_Stellung_2;
      );
      JC    disp;
// 2 ==> grau
      L     2;
      AN    #io_Stoerung;
      A(;
      AN    DIX [AR2,P#0.5];	// Kennung "invers"
//      UN    #in_Eingang_Stellung_1    // (016)
      A     #in_Eingang_Stellung_1;	// (016)
//      U     #in_Eingang_Stellung_2    // (016)
      AN    #in_Eingang_Stellung_2;	// (016)
      AN    #io_Ausgang_Stellung_1;
//      U     #io_Ausgang_Stellung_2    // (016)
      AN    #io_Ausgang_Stellung_2;	// (016)
      O;
      A     DIX [AR2,P#0.5];	// Kennung "invers"
//      U     #in_Eingang_Stellung_1    // (016)
      AN    #in_Eingang_Stellung_1;	// (016)
//      UN    #in_Eingang_Stellung_2    // (016)
      A     #in_Eingang_Stellung_2;	// (016)
//      U     #io_Ausgang_Stellung_1    // (016)
      AN    #io_Ausgang_Stellung_1;	// (016)
      AN    #io_Ausgang_Stellung_2;
      );
      JC    disp;
// 5 ==> grün
      L     5;
      AN    #io_Stoerung;
      A(;
      AN    DIX [AR2,P#0.5];	// Kennung "invers"
//      U     #in_Eingang_Stellung_1    // (016)
      AN    #in_Eingang_Stellung_1;	// (016)
//      UN    #in_Eingang_Stellung_2    // (016)
      A     #in_Eingang_Stellung_2;	// (016)
      AN    #io_Ausgang_Stellung_1;
//      UN    #io_Ausgang_Stellung_2    // (016)
      A     #io_Ausgang_Stellung_2;	// (016)
      O;
      A     DIX [AR2,P#0.5];	// Kennung "invers"
//      UN    #in_Eingang_Stellung_1    // (016)
      A     #in_Eingang_Stellung_1;	// (016)
//      U     #in_Eingang_Stellung_2    // (016)
      AN    #in_Eingang_Stellung_2;	// (016)
//      UN    #io_Ausgang_Stellung_1    // (016)
      A     #io_Ausgang_Stellung_1;	// (016)
      AN    #io_Ausgang_Stellung_2;
      );
      JC    disp;
// 6 ==> grün
      L     6;
      AN    #io_Stoerung;
      A(;
      AN    DIX [AR2,P#0.5];	// Kennung "invers"
      A     #in_Eingang_Stellung_1;
      AN    #in_Eingang_Stellung_2;
      A     #io_Ausgang_Stellung_1;
      AN    #io_Ausgang_Stellung_2;
      O;
      A     DIX [AR2,P#0.5];	// Kennung "invers"
      AN    #in_Eingang_Stellung_1;
      A     #in_Eingang_Stellung_2;
      AN    #io_Ausgang_Stellung_1;
      A     #io_Ausgang_Stellung_2;
      );
      JC    disp;
// 9 ==> weiß
      L     9;
      AN    #io_Stoerung;
      A(;
      AN    DIX [AR2,P#0.5];	// Kennung "invers"
      AN    #in_Eingang_Stellung_1;
      AN    #in_Eingang_Stellung_2;
      AN    #io_Ausgang_Stellung_1;
      A     #io_Ausgang_Stellung_2;
      O;
      A     DIX [AR2,P#0.5];	// Kennung "invers"
      AN    #in_Eingang_Stellung_1;
      AN    #in_Eingang_Stellung_2;
      A     #io_Ausgang_Stellung_1;
      AN    #io_Ausgang_Stellung_2;
      );
      JC    disp;
// 10 ==> weiß
      L     10;
      AN    #io_Stoerung;
      A(;
      AN    DIX [AR2,P#0.5];	// Kennung "invers"
      AN    #in_Eingang_Stellung_1;
      AN    #in_Eingang_Stellung_2;
      A     #io_Ausgang_Stellung_1;
      AN    #io_Ausgang_Stellung_2;
      O;
      A     DIX [AR2,P#0.5];	// Kennung "invers"
      AN    #in_Eingang_Stellung_1;
      AN    #in_Eingang_Stellung_2;
      AN    #io_Ausgang_Stellung_1;
      A     #io_Ausgang_Stellung_2;
      );
      JC    disp;
// 11 ==> hellgrün
      L     11;
      A     DIX [AR2,P#1.2];	// Kennung "grob/fein"
      A     #io_Ausgang_Stellung_1;
      A     #io_Ausgang_Stellung_2;
      AN    #in_Eingang_Stellung_1;
      AN    #in_Eingang_Stellung_2;
      AN    #io_Stoerung;
      JC    disp;
// 14 = Störung, quittierpflichtig, Ausgang nicht angesteuert, Störung ==> rot/weiß
      L     14;	// (014)
      A     #io_Stoerung;	// (014)
      AN    #in_Quitt_Stoerung;	// (014)
      AN    #io_Ausgang_Stellung_1;	// (014)
      AN    #io_Ausgang_Stellung_2;	// (014)
      JC    disp;	// (014)
// 15 = Störung, nicht quittierpflichtig, Ausgang angesteuert, Störung ==> rot/grün
      L     15;	// (014)
      A     #io_Stoerung;	// (014)
      AN    #in_Quitt_Stoerung;	// (014)
      A(;	// (014)
      O     #io_Ausgang_Stellung_1;	// (014)
      O     #io_Ausgang_Stellung_2;	// (014)
      );	// (014)
      JC    disp;	// (014)
// 16 = Störung quittiert ==> rot
      L     16;
      A     #io_Stoerung;
      JC    disp;
NSV2: NOP   0;
NETWORK
TITLE = Objektstatus für Visualisation OP (011)(012)(017)
//Stati:
//-------
//1 = Eingang Position 2, keine Störung ==> grau
//5 = Eingang Position 1, keine Störung ==> grün
//9 = nicht Eingang 1 und nicht Eingang 2, keine Störung ==> weiß
//14 = Störung, Stellung 2, nicht quittiert ==> rot/weiß
//15 = Störung, Stellung 1, nicht quittiert ==> rot/grün
//16 = Störung quittiert ==> rot
      A(;
      O     DIX [AR2,P#0.6];	// Kennung "auf/zu"
      O     DIX [AR2,P#1.1];	// Kennung "oben/unten" // (022)
      O     DIX [AR2,P#1.3];	// Kennung "ein/aus"
      O     DIX [AR2,P#1.4];	// Kennung "spannen/lösen"
      O     DIX [AR2,P#1.5];	// Kennung "andocken/abdocken"
      O     DIX [AR2,P#1.7];	// Kennung "vor/zurück"   // (022)
      );
      JCN   NSV3;	// Not Status Version 3
// 1 ==> grau
      L     1;
      AN    #io_Stoerung;
      A(;
      AN    DIX [AR2,P#0.5];	// Kennung "invers"
      A     #in_Eingang_Stellung_2;
      O;
      A     DIX [AR2,P#0.5];	// Kennung "invers"
      A     #in_Eingang_Stellung_1;
      );
      JC    disp;
// 6 ==> grün
      L     6;	// (019) = besser weil Fehlertoleranter als 5
      AN    #io_Stoerung;
      A(;
      AN    DIX [AR2,P#0.5];	// Kennung "invers"
      A     #in_Eingang_Stellung_1;
      O;
      A     DIX [AR2,P#0.5];	// Kennung "invers"
      A     #in_Eingang_Stellung_2;
      );
      JC    disp;
// 9 ==> weiß
      L     9;
      AN    #io_Stoerung;
      A(;
      AN    DIX [AR2,P#0.5];	// Kennung "invers"
      AN    #in_Eingang_Stellung_1;
      AN    #in_Eingang_Stellung_2;
      O;
      A     DIX [AR2,P#0.5];	// Kennung "invers"
      AN    #in_Eingang_Stellung_1;
      AN    #in_Eingang_Stellung_2;
      );
      JC    disp;
// 14 = Störung, Stellung 2, nicht quittiert ==> rot/weiß
      L     14;
      A     #io_Stoerung;
      AN    #in_Quitt_Stoerung;
      A(;
      AN    DIX [AR2,P#0.5];	// Kennung "invers"
      AN    #in_Eingang_Stellung_1;	// (018) = Stellung 2 oder Keine
      O;
      A     DIX [AR2,P#0.5];	// Kennung "invers"
      AN    #in_Eingang_Stellung_2;	// (018) = Stellung 1 oder Keine
      );
      JC    disp;
// 15 = Störung, Stellung 1, nicht quittiert ==> rot/grün
      L     15;
      A     #io_Stoerung;
      AN    #in_Quitt_Stoerung;
      A(;
      AN    DIX [AR2,P#0.5];	// Kennung "invers"
      A     #in_Eingang_Stellung_1;
      O;
      A     DIX [AR2,P#0.5];	// Kennung "invers"
      A     #in_Eingang_Stellung_2;
      );
      JC    disp;
// 16 = Störung quittiert ==> rot
      L     16;
      A     #io_Stoerung;
      JC    disp;
NSV3: NOP   0;
NETWORK
TITLE = Objektstatus speichern (017)
//jm 20120907
      L     0;
disp: T     #Objektstatus;
NETWORK
TITLE = Daten in Struktur speichern
      A     #in_Anlage_ein;	// (021)
      =     DIX [AR2,P#4.5];	// (021) Anlage ein (Struktur)
      A     #in_Eingang_Stellung_1;
      =     DIX [AR2,P#2.2];	// Eingang Stellung 1 (Struktur)
      A     #in_Eingang_Stellung_2;
      =     DIX [AR2,P#2.3];	// Eingang Stellung 2 (Struktur)
      A     #io_Ausgang_Stellung_1;
      =     DIX [AR2,P#2.0];	// Ausgang Stellung 1 (Struktur)
      A     #io_Ausgang_Stellung_2;
      =     DIX [AR2,P#2.1];	// Ausgang Stellung 2 (Struktur)
      A     #io_Stellung_1_Betrieb;
      =     DIX [AR2,P#2.6];	// Stellung 1 in Betrieb (Struktur)
      A     #io_Stellung_2_Betrieb;
      =     DIX [AR2,P#2.7];	// Stellung 2 in Betrieb (Struktur)
      A     #io_Stoerung;
      =     DIX [AR2,P#3.0];	// Störung (Struktur)
      A     #Taktanzahl_erreicht;
      =     DIX [AR2,P#3.7];	// Taktanzahl erreicht (Struktur)
      A     #Taktausgang;
      =     DIX [AR2,P#4.3];	// Taktausgang (Struktur)
      L     #Zeitzaehler;
      T     DID [AR2,P#18.0];	// Impuls-/Pausezähler (Struktur)
      L     #Taktzaehler;
      T     DIW [AR2,P#24.0];	// Taktzähler (Struktur)
      L     #Objektstatus;	// (011)
      T     DIW [AR2,P#48.0];	// #Objektstatus  (Struktur)   // (011)
NETWORK
TITLE = ENDE
      NOP   0;
END_FUNCTION

FUNCTION "FC23 Ventil 1-10A" : VOID	// FC 23
TITLE = Bock for actuating several cycled valves
//Erstellung:
//Datum       Bearbeiter                                                   Version
//--------------------------------------------------------------------------------
//14.06.99    A.Kirchgessner(kia)                                         01.00.00
//
//Änderungen:
//Nr. Datum    Bearb Änderung                                       Marke  Version
//--------------------------------------------------------------------------------
//01  16.07.99 kia   Fehlerbeseitigung                                    01.00.01
//02  12.08.99 sra   Fehlerbeseitigung mit Parameteränderung              01.01.00
//03  19.10.99 sra   Anpassung an neue Struktur                           01.02.00
//04  10.07.00 sra   Fehlerbeseitigung Taktgenerierung                    01.02.01
//05  10.07.00 sra   Änderung in Eingangsparameter                        01.03.00
//06  19.09.00 sra   komplette Überarbeitung / neue Struktur              02.00.00
//07  18.01.01 gea   Erweiterung auf 10 Ventile / neue Struktur           02.01.00
//08  27.03.02 sra   Meldung "Ventil in Betrieb" auch im Handmode   (008) 02.01.01
//09  04.02.03 kal   Fehlerbeseitigung Dauertakt                    (009) 02.01.02
//10  31.10.05 sra   Ansteuerung Handbedienung im Automode rücksetz.
//                   Handbedienung zentral sperren                  (010) 02.02.00
//11  18.02.09 kmj   Objektststatus für OP ergänzt                  (011) 02.03.00
//12  20.03.09 kal   Objektststatus für OP ergänzt (überarbeitet)   (012) 02.03.01
//13  24.04.09 gea   Handmode zurücksetzen wenn Handmode gesperrt   (013) 02.03.02
//14  05.12.13 sra   "Anlage ein" eingefügt (Not-Aus-Konzept)       (014) 02.04.00
//15  14.11.14 bhl   Anzeige "#io_Ventil_in_Betrieb" im Handmode    (015) 02.04.01
//16  11.08.15 sra   "#io_Ventil_in_Betrieb" nur wenn "Anlage ein"  (016) 02.04.02
//________________________________________________________________________________
//Eingesetzte Bausteine:
//
//FC2 : Version 01.01.XX
//________________________________________________________________________________
//Funktion:
//
//Der Baustein taktet die einzelnen Ventile der Reihe nach durch (Anzahl der 
//Ventile max. 10 Stück). 
//
//Die Ausgänge werden nur angesteuert wenn der Eingang "in_Anlage_ein" = true
//ist. Diese Funktion ist vorhanden, um bei einem Not-Halt die Anlage vor 
//unkontrolliertem Einschalten zu schützen. 
//
//Im Handmode werden die ausgewählten Ventile dauerhaft angesteuert. 
//
AUTHOR : kia
FAMILY : AZO
VERSION : 0.0
VAR_INPUT
  in_Handbedienung_erlaubt : BOOL ;	//1 = manual operation permitted, 0 = manual operation not permitted/locked
  in_Anlage_ein : BOOL ;	//Anlage bzw. Anlagenbereich nach Not-Halt freigegeben
  in_Ansteuerung_Ventil_T1 : BOOL ;	//Actuation of valve position 1 in automatic mode with cycle 1
  in_Ansteuerung_Ventil_T2 : BOOL ;	//Actuation of valve position 1 in automatic mode with cycle 2
END_VAR
VAR_IN_OUT
  io_Ausgang_Ventil_1 : BOOL ;	//Output 1. Valve
  io_Ausgang_Ventil_2 : BOOL ;	//Output 2. Valve
  io_Ausgang_Ventil_3 : BOOL ;	//Output 3. Valve
  io_Ausgang_Ventil_4 : BOOL ;	//Output 4. Valve
  io_Ausgang_Ventil_5 : BOOL ;	//Output 5. Valve
  io_Ausgang_Ventil_6 : BOOL ;	//Output 6. Valve
  io_Ausgang_Ventil_7 : BOOL ;	//Output 7. Valve
  io_Ausgang_Ventil_8 : BOOL ;	//Output 8. Valve
  io_Ausgang_Ventil_9 : BOOL ;	//Output 9. Valve
  io_Ausgang_Ventil_10 : BOOL ;	//Output 10. Valve
  io_Ventil_in_Betrieb : BOOL ;	//Signal "valve in operation" (actuated)
  io_Ventilstruktur : ANY ;	//ANY pointer of valve structure
END_VAR
VAR_TEMP
  Ventilansteuerung : BOOL ;	//Freigabe ein Ventil anzusteuern
  Freigabe_Takt : BOOL ;	//Cycle enable
  Rueckmeldung : BOOL ;	//wenn eines der Ventil agesteuert ist --> 1-Signal
  Start_mit_Impuls : BOOL ;
  Taktanzahl_erreicht : BOOL ;
  Dauertakt : BOOL ;	//Continuous cycle
  positive_Flanke : BOOL ;
  Hilfs_Anzahl_Takte : INT ;	//Sollvorgabe für FC2
  Aktuelles_Ventil : INT ;	//aktuelles Ventil
  Hilfswort_1 : INT ;
  Impulszeit_Takt : REAL ;
  Pausezeit_Takt : REAL ;
  Zeitzaehler : REAL ;
  Taktzaehler : INT ;
  Objektstatus : INT ;
END_VAR
BEGIN
NETWORK
TITLE = Anfangs-DW der Struktur aus ANY-Zeiger auslesen
      L     P##io_Ventilstruktur;
      LAR2;
      L     D [AR2,P#6.0];
      LAR2;	//Pointer auf Structuranfang
NETWORK
TITLE = Umschaltung Hand-/Automatikmode 
      A     DIX [AR2,P#3.6];	// Handmode von Farbgrafik (Struktur)
      AN    DIX [AR2,P#5.1];	// Handmode gesperrt (Struktur)
      AN    "M0.0 LockManualMode";	// Handbedienung zentral sperren (010)
      S     DIX [AR2,P#3.5];	// Handmode zu Farbgrafik (Struktur)
      ON    DIX [AR2,P#3.6];	// Handmode von Farbgrafik (Struktur)
      ON    #in_Handbedienung_erlaubt;
      O     "M0.0 LockManualMode";	// Handbedienung zentral sperren (010)
      O     DIX [AR2,P#5.1];	// Handmode gesperrt (Struktur) (013)
      R     DIX [AR2,P#3.5];	// Handmode zu Farbgrafik (Struktur)
      R     DIX [AR2,P#3.6];	// Handmode von Farbgrafik (Struktur) (010)
NETWORK
TITLE = Ansteuerung Handmode zurücksetzen
//(010) 
      AN    DIX [AR2,P#3.5];	// Handmode zu Farbgrafik (Struktur)
      R     DIX [AR2,P#3.7];	// Ansteuerung des 1. Ventils im Handmode von Farbgrafik (Struktur)
      R     DIX [AR2,P#4.0];	// Ansteuerung des 2. Ventils im Handmode von Farbgrafik (Struktur)
      R     DIX [AR2,P#4.1];	// Ansteuerung des 3. Ventils im Handmode von Farbgrafik (Struktur)
      R     DIX [AR2,P#4.2];	// Ansteuerung des 4. Ventils im Handmode von Farbgrafik (Struktur)
      R     DIX [AR2,P#4.3];	// Ansteuerung des 5. Ventils im Handmode von Farbgrafik (Struktur)
      R     DIX [AR2,P#4.4];	// Ansteuerung des 6. Ventils im Handmode von Farbgrafik (Struktur)
      R     DIX [AR2,P#4.5];	// Ansteuerung des 7. Ventils im Handmode von Farbgrafik (Struktur)
      R     DIX [AR2,P#4.6];	// Ansteuerung des 8. Ventils im Handmode von Farbgrafik (Struktur)
      R     DIX [AR2,P#4.7];	// Ansteuerung des 9. Ventils im Handmode von Farbgrafik (Struktur)
      R     DIX [AR2,P#5.0];	// Ansteuerung des 10. Ventils im Handmode von Farbgrafik (Struktur)
NETWORK
TITLE = Rueckmeldung Ventile + Ventilansteuerung
      O     #io_Ausgang_Ventil_1;
      O     #io_Ausgang_Ventil_2;
      O     #io_Ausgang_Ventil_3;
      O     #io_Ausgang_Ventil_4;
      O     #io_Ausgang_Ventil_5;
      O     #io_Ausgang_Ventil_6;
      O     #io_Ausgang_Ventil_7;
      O     #io_Ausgang_Ventil_8;
      O     #io_Ausgang_Ventil_9;
      O     #io_Ausgang_Ventil_10;
      =     #Rueckmeldung;
      =     #Ventilansteuerung;
NETWORK
TITLE = Daten für Takt in temporäre Variablen laden
//(009) komplettes Netzwerk gelöscht.
//Dauertakt nur, wenn Bit in Struktur = TRUE 
//Anzahl Takte ist egal!!!
      A     DIX [AR2,P#5.2];	// Start mit Impuls (Struktur)
      =     #Start_mit_Impuls;
      A     DIX [AR2,P#5.3];	// Taktanzahl erreicht (Struktur)
      =     #Taktanzahl_erreicht;
      A     DIX [AR2,P#5.4];	// Dauertakt (Struktur)
      =     #Dauertakt;
      L     DID [AR2,P#22.0];	// Impuls-/Pausezähler (Struktur)
      T     #Zeitzaehler;
      L     DIW [AR2,P#28.0];	// Taktzähler (Struktur)
      T     #Taktzaehler;
NETWORK
TITLE = Sollanzahl Takte
      AN    #Dauertakt;
      JC    ST_1;
      L     DIW [AR2,P#30.0];	// Anzahl Ventile (Struktur)
      T     #Hilfs_Anzahl_Takte;
ST_1: NOP   0;
      A     #Dauertakt;
      JC    ST_2;
      L     DIW [AR2,P#26.0];	// Sollanzahl Takte (Struktur)
      T     #Hilfs_Anzahl_Takte;
ST_2: NOP   0;
NETWORK
TITLE = Freigabe Takt
      A     #in_Anlage_ein;	// (014)
      A(;	// (014)
      O     #in_Ansteuerung_Ventil_T1;
      O     #in_Ansteuerung_Ventil_T2;
      );	// (014)
      =     #Freigabe_Takt;
NETWORK
TITLE = Takt umkopieren
      L     DID [AR2,P#6.0];	// Impulszeit Befüllung (Struktur)
      T     #Impulszeit_Takt;
      L     DID [AR2,P#10.0];	// Pausezeit Befüllung (Struktur)
      T     #Pausezeit_Takt;
      A     #in_Ansteuerung_Ventil_T1;
      JC    E_Tk;
      L     DID [AR2,P#14.0];	// Impulszeit Entleerung (Struktur)
      T     #Impulszeit_Takt;
      L     DID [AR2,P#18.0];	// Pausezeit Entleerung (Struktur)
      T     #Pausezeit_Takt;
E_Tk: NOP   0;
NETWORK
TITLE = Takt generieren
      CALL  "FC2 Taktgeber_Timernachb" (
           in_Freigabe              := #Freigabe_Takt,
           in_Rueckmeldung          := #Rueckmeldung,
           in_Start_mit_Impuls      := #Start_mit_Impuls,
           in_Dauertakt             := #Dauertakt,
           in_Impuls                := "M1.7 ClockTimerFunction",
           in_Impulszeit_in_100ms   := "MW 6 Timer Val Cycle FCs",
           in_Impulszeit            := #Impulszeit_Takt,
           in_Pausezeit             := #Pausezeit_Takt,
           in_Sollanzahl_Takte      := #Hilfs_Anzahl_Takte,
           io_Taktausgang           := #Ventilansteuerung,
           io_Taktanzahl_erreicht   := #Taktanzahl_erreicht,
           io_Zeitzaehler           := #Zeitzaehler,
           io_Taktzaehler           := #Taktzaehler);
NETWORK
TITLE = aktuelles Ventil
      L     #Taktzaehler;
      L     DIW [AR2,P#30.0];	// Anzahl Ventile (Struktur)
      /I;
      T     #Hilfswort_1;
      L     #Hilfswort_1;
      L     DIW [AR2,P#30.0];	// Anzahl Ventile (Struktur)
      *I;
      L     -1;
      *I;
      L     #Taktzaehler;
      +I;
      L     1;
      +I;
      T     #Aktuelles_Ventil;
NETWORK
TITLE = aktuelles Ventil prüfen
      A(;
      L     #Aktuelles_Ventil;
      L     1;
      >=I;
      );
      A(;
      L     #Aktuelles_Ventil;
      L     DIW [AR2,P#30.0];	// Anzahl Ventile (Struktur)
      <=I;
      );
      JC    M1;
      L     1;
      T     #Aktuelles_Ventil;
M1:   NOP   0;
NETWORK
TITLE = Ansteuerung Ventil 1
      A     #in_Anlage_ein;	// (014)
      A(;	// (014)
      A(;
      L     #Aktuelles_Ventil;
      L     1;
      ==I;
      );
      A(;	// Automatikmode
      AN    DIX [AR2,P#3.5];	// Handmode zu Farbgrafik (Struktur)
      A     #Ventilansteuerung;
      AN    #Taktanzahl_erreicht;
      );
      O;	// Handmode 
      A     DIX [AR2,P#3.5];	// Handmode zu Farbgrafik (Struktur)
      A     DIX [AR2,P#3.7];	// Ansteuerung des 1. Ventils im Handmode von Farbgrafik (Struktur)
      );	// (014)
      =     #io_Ausgang_Ventil_1;
NETWORK
TITLE = Ansteuerung Ventil 2
      A     #in_Anlage_ein;	// (014)
      A(;	// (014)
      A(;
      L     #Aktuelles_Ventil;
      L     2;
      ==I;
      );
      A(;	// Automatikmode
      AN    DIX [AR2,P#3.5];	// Handmode zu Farbgrafik (Struktur)
      A     #Ventilansteuerung;
      AN    #Taktanzahl_erreicht;
      );
      O;	// Handmode 
      A     DIX [AR2,P#3.5];	// Handmode zu Farbgrafik (Struktur)
      A     DIX [AR2,P#4.0];	// Ansteuerung des 2. Ventils im Handmode von Farbgrafik (Struktur)
      );	// (014)
      =     #io_Ausgang_Ventil_2;
NETWORK
TITLE = Ansteuerung Ventil 3
      A     #in_Anlage_ein;	// (014)
      A(;	// (014)
      A(;
      L     #Aktuelles_Ventil;
      L     3;
      ==I;
      );
      A(;	// Automatikmode
      AN    DIX [AR2,P#3.5];	// Handmode zu Farbgrafik (Struktur)
      A     #Ventilansteuerung;
      AN    #Taktanzahl_erreicht;
      );
      O;	// Handmode 
      A     DIX [AR2,P#3.5];	// Handmode zu Farbgrafik (Struktur)
      A     DIX [AR2,P#4.1];	// Ansteuerung des 3. Ventils im Handmode von Farbgrafik (Struktur)
      );	// (014)
      =     #io_Ausgang_Ventil_3;
NETWORK
TITLE = Ansteuerung Ventil 4
      A     #in_Anlage_ein;	// (014)
      A(;	// (014)
      A(;
      L     #Aktuelles_Ventil;
      L     4;
      ==I;
      );
      A(;	// Automatikmode
      AN    DIX [AR2,P#3.5];	// Handmode zu Farbgrafik (Struktur)
      A     #Ventilansteuerung;
      AN    #Taktanzahl_erreicht;
      );
      O;	// Handmode 
      A     DIX [AR2,P#3.5];	// Handmode zu Farbgrafik (Struktur)
      A     DIX [AR2,P#4.2];	// Ansteuerung des 4. Ventils im Handmode von Farbgrafik (Struktur)
      );	// (014)
      =     #io_Ausgang_Ventil_4;
NETWORK
TITLE = Ansteuerung Ventil 5
      A     #in_Anlage_ein;	// (014)
      A(;	// (014)
      A(;
      L     #Aktuelles_Ventil;
      L     5;
      ==I;
      );
      A(;	// Automatikmode
      AN    DIX [AR2,P#3.5];	// Handmode zu Farbgrafik (Struktur)
      A     #Ventilansteuerung;
      AN    #Taktanzahl_erreicht;
      );
      O;	// Handmode 
      A     DIX [AR2,P#3.5];	// Handmode zu Farbgrafik (Struktur)
      A     DIX [AR2,P#4.3];	// Ansteuerung des 5. Ventils im Handmode von Farbgrafik (Struktur)
      );	// (014)
      =     #io_Ausgang_Ventil_5;
NETWORK
TITLE = Ansteuerung Ventil 6
      A     #in_Anlage_ein;	// (014)
      A(;	// (014)
      A(;
      L     #Aktuelles_Ventil;
      L     6;
      ==I;
      );
      A(;	// Automatikmode
      AN    DIX [AR2,P#3.5];	// Handmode zu Farbgrafik (Struktur)
      A     #Ventilansteuerung;
      AN    #Taktanzahl_erreicht;
      );
      O;	// Handmode 
      A     DIX [AR2,P#3.5];	// Handmode zu Farbgrafik (Struktur)
      A     DIX [AR2,P#4.4];	// Ansteuerung des 6. Ventils im Handmode von Farbgrafik (Struktur)
      );	// (014)
      =     #io_Ausgang_Ventil_6;
NETWORK
TITLE = Ansteuerung Ventil 7
      A     #in_Anlage_ein;	// (014)
      A(;	// (014)
      A(;
      L     #Aktuelles_Ventil;
      L     7;
      ==I;
      );
      A(;	// Automatikmode
      AN    DIX [AR2,P#3.5];	// Handmode zu Farbgrafik (Struktur)
      A     #Ventilansteuerung;
      AN    #Taktanzahl_erreicht;
      );
      O;	// Handmode 
      A     DIX [AR2,P#3.5];	// Handmode zu Farbgrafik (Struktur)
      A     DIX [AR2,P#4.5];	// Ansteuerung des 7. Ventils im Handmode von Farbgrafik (Struktur)
      );	// (014)
      =     #io_Ausgang_Ventil_7;
NETWORK
TITLE = Ansteuerung Ventil 8
      A     #in_Anlage_ein;	// (014)
      A(;	// (014)
      A(;
      L     #Aktuelles_Ventil;
      L     8;
      ==I;
      );
      A(;	// Automatikmode
      AN    DIX [AR2,P#3.5];	// Handmode zu Farbgrafik (Struktur)
      A     #Ventilansteuerung;
      AN    #Taktanzahl_erreicht;
      );
      O;	// Handmode 
      A     DIX [AR2,P#3.5];	// Handmode zu Farbgrafik (Struktur)
      A     DIX [AR2,P#4.6];	// Ansteuerung des 8. Ventils im Handmode von Farbgrafik (Struktur)
      );	// (014)
      =     #io_Ausgang_Ventil_8;
NETWORK
TITLE = Ansteuerung Ventil 9
      A     #in_Anlage_ein;	// (014)
      A(;	// (014)
      A(;
      L     #Aktuelles_Ventil;
      L     9;
      ==I;
      );
      A(;	// Automatikmode
      AN    DIX [AR2,P#3.5];	// Handmode zu Farbgrafik (Struktur)
      A     #Ventilansteuerung;
      AN    #Taktanzahl_erreicht;
      );
      O;	// Handmode 
      A     DIX [AR2,P#3.5];	// Handmode zu Farbgrafik (Struktur)
      A     DIX [AR2,P#4.7];	// Ansteuerung des 9. Ventils im Handmode von Farbgrafik (Struktur)
      );	// (014)
      =     #io_Ausgang_Ventil_9;
NETWORK
TITLE = Ansteuerung Ventil 10
      A     #in_Anlage_ein;	// (014)
      A(;	// (014)
      A(;
      L     #Aktuelles_Ventil;
      L     10;
      ==I;
      );
      A(;	// Automatikmode
      AN    DIX [AR2,P#3.5];	// Handmode zu Farbgrafik (Struktur)
      A     #Ventilansteuerung;
      AN    #Taktanzahl_erreicht;
      );
      O;	// Handmode 
      A     DIX [AR2,P#3.5];	// Handmode zu Farbgrafik (Struktur)
      A     DIX [AR2,P#5.0];	// Ansteuerung des 10. Ventils im Handmode von Farbgrafik (Struktur)
      );	// (014)
      =     #io_Ausgang_Ventil_10;
NETWORK
TITLE = Ausgang Betrieb
      AN    DIX [AR2,P#3.5];	// (015) Handmode zu Farbgrafik (Struktur)
      A     #in_Anlage_ein;	// (016)
      A(;
      O     #in_Ansteuerung_Ventil_T1;
      O     #in_Ansteuerung_Ventil_T2;	// (008)
      );
      A     #Dauertakt;
      O;
      AN    DIX [AR2,P#3.5];	// (015) Handmode zu Farbgrafik (Struktur)
      A     #in_Anlage_ein;	// (016)
      A(;
      O     #in_Ansteuerung_Ventil_T1;
      O     #in_Ansteuerung_Ventil_T2;
      );
      AN    #Dauertakt;
      AN    #Taktanzahl_erreicht;
      O;
      A     DIX [AR2,P#3.5];	// Handmode zu Farbgrafik (Struktur)
      A     #in_Anlage_ein;	// (016)
      A(;
      O     #io_Ausgang_Ventil_1;	// (008)
      O     #io_Ausgang_Ventil_2;	// (008)
      O     #io_Ausgang_Ventil_3;	// (008)
      O     #io_Ausgang_Ventil_4;	// (008)
      O     #io_Ausgang_Ventil_5;	// (008)
      O     #io_Ausgang_Ventil_6;	// (008)
      O     #io_Ausgang_Ventil_7;	// (008)
      O     #io_Ausgang_Ventil_8;	// (008)
      O     #io_Ausgang_Ventil_9;	// (008)
      O     #io_Ausgang_Ventil_10;	// (008)
      );
      =     #io_Ventil_in_Betrieb;
NETWORK
TITLE = Flankenauswertung Ausgang Ventil für Schalthäufigkeitzähler
//Es wird die Schalthäufigkeit der Ventile gezählt !  
      O     #io_Ausgang_Ventil_1;
      O     #io_Ausgang_Ventil_2;
      O     #io_Ausgang_Ventil_3;
      O     #io_Ausgang_Ventil_4;
      O     #io_Ausgang_Ventil_5;
      O     #io_Ausgang_Ventil_6;
      O     #io_Ausgang_Ventil_7;
      O     #io_Ausgang_Ventil_8;
      O     #io_Ausgang_Ventil_9;
      O     #io_Ausgang_Ventil_10;
      FP    DIX [AR2,P#32.3];	// Flankenmerker Ausgang (Struktur)
      =     #positive_Flanke;
NETWORK
TITLE = Schalthäufigkeitzähler
      ON    DIX [AR2,P#0.3];	// Kennung Schalthäufigkeitzähler ein (Struktur)
      ON    #positive_Flanke;
      JC    ESHZ;
      L     1.000000e+00;
      L     DID [AR2,P#34.0];	// Schalthäufigkeitzähler (Struktur)
      +R;
      T     DID [AR2,P#34.0];	// Schalthäufigkeitzähler (Struktur)
ESHZ: NOP   0;
NETWORK
TITLE = Schalthäufigkeitzähler zurücksetzten
      AN    DIX [AR2,P#32.0];	// Reset Schalthäufigkeitzähler (Struktur)
      JC    E_RS;
      L     0.000000e+00;
      T     DID [AR2,P#34.0];	// Schalthäufigkeitzähler (Struktur)
      CLR;
      =     DIX [AR2,P#32.0];	// Reset Schalthäufigkeitzähler (Struktur)
E_RS: NOP   0;
NETWORK
TITLE = Warnmeldung Schalthäufigkeitzähler erzeugen
      A(;
      L     DID [AR2,P#34.0];	// Schalthäufigkeitzähler (Struktur)
      L     DID [AR2,P#38.0];	// Sollwert Warnung (Struktur)
      >R;
      );
      A(;
      L     DID [AR2,P#38.0];	// Sollwert Warnung (Struktur)
      L     0.000000e+00;
      <>R;
      );
      =     DIX [AR2,P#32.1];	// Warnmeldung Schalthäufigkeitzähler (Struktur)
NETWORK
TITLE = Alarmmeldung Schalthäufigkeitzähler erzeugen
      A(;
      L     DID [AR2,P#34.0];	// Schalthäufigkeitzähler (Struktur)
      L     DID [AR2,P#42.0];	// Sollwert Alarm (Struktur)
      >R;
      );
      A(;
      L     DID [AR2,P#42.0];	// Sollwert Alarm (Struktur)
      L     0.000000e+00;
      <>R;
      );
      =     DIX [AR2,P#32.2];	// Warnmeldung Schalthäufigkeitzähler (Struktur)
NETWORK
TITLE = Objektstatus für Visualisation OP (011)(012)
//Stati:
//-------
//1 = kein Ventil angesteuert ==> Farbvorschlag weiß
//5 = ein ventil in Betrieb ==> Farbvorschlag grün
//
// 1 = nicht in Betrieb, keine Störung ==> Farbvorschlag grau
      L     1;
      AN    #io_Ventil_in_Betrieb;
      JC    disp;
// 5 = angesteuert, nicht in Betrieb, keine Störung ==> Farbvorschlag grün
      L     5;
      A     #io_Ventil_in_Betrieb;
      JC    disp;
      L     0;
disp: T     #Objektstatus;
NETWORK
TITLE = Daten in Struktur speichern
      A     #in_Anlage_ein;	// (014)
      =     DIX [AR2,P#5.5];	// (014) Anlage ein (Struktur)
      A     #io_Ausgang_Ventil_1;
      =     DIX [AR2,P#2.0];	// Ausgang Ventil 1 (Struktur)
      A     #io_Ausgang_Ventil_2;
      =     DIX [AR2,P#2.1];	// Ausgang Ventil 2 (Struktur)
      A     #io_Ausgang_Ventil_3;
      =     DIX [AR2,P#2.2];	// Ausgang Ventil 3 (Struktur)
      A     #io_Ausgang_Ventil_4;
      =     DIX [AR2,P#2.3];	// Ausgang Ventil 4 (Struktur)
      A     #io_Ausgang_Ventil_5;
      =     DIX [AR2,P#2.4];	// Ausgang Ventil 5 (Struktur)
      A     #io_Ausgang_Ventil_6;
      =     DIX [AR2,P#2.5];	// Ausgang Ventil 6 (Struktur)
      A     #io_Ausgang_Ventil_7;
      =     DIX [AR2,P#2.6];	// Ausgang Ventil 7 (Struktur)
      A     #io_Ausgang_Ventil_8;
      =     DIX [AR2,P#2.7];	// Ausgang Ventil 8 (Struktur)
      A     #io_Ausgang_Ventil_9;
      =     DIX [AR2,P#3.0];	// Ausgang Ventil 9 (Struktur)
      A     #io_Ausgang_Ventil_10;
      =     DIX [AR2,P#3.1];	// Ausgang Ventil 10 (Struktur)
      A     #io_Ventil_in_Betrieb;
      =     DIX [AR2,P#3.4];	// Ventil in Betrieb (Struktur)
      A     #Taktanzahl_erreicht;
      =     DIX [AR2,P#5.3];	// Taktanzahl erreicht (Struktur)
      L     #Zeitzaehler;
      T     DID [AR2,P#22.0];	// Impuls-/Pausezähler (Struktur)
      L     #Taktzaehler;
      T     DIW [AR2,P#28.0];	// Taktzähler (Struktur)
      L     #Objektstatus;	// (011)
      T     DIW [AR2,P#48.0];	// #Objektstatus  (Struktur)   // (011)
END_FUNCTION

FUNCTION "FC24 Binär-E" : VOID	// FC 24
TITLE = Block for debouncing and fault monitoring of a binary input
//Building:
//Date         Editor                                                     Version
//--------------------------------------------------------------------------------
//22.09.99     (jm)                                                       01.00.00
//
//Modifications:
//No. Date     Edit  Description                                    Index Version
//--------------------------------------------------------------------------------
//01  29.09.00 sra   komplette Überarbeitung / neue Struktur        ()    02.00.00
//02  16.06.05 sra   Änderung INC 1 -> + 1                         (002)  02.00.01
//03  04.09.06 sra   Änderung Störungsquittierung                  (003)  02.01.00
//04  08.07.10 jm    Störzeit 0 möglich                            (004)  02.01.01
//05  06.06.16 kal/sra komplette Überarbeitung (wie TIA-Portal)     ()    03.00.00
//06  12.06.16 sra   Änderung Signal "Eingang verarbeitet"         (006)  03.01.00
//07  13.12.17 gea   Objektstatus betätig/störung (neu)            (007)  03.02.00
//                   Objektstatus nicht betätig/störung (neu)
//                   Eingang verarbeitet bei Störung ausgeben
//08  26.01.18 gea   Objektstatus Fehlerbeseitigung                (008)  03.02.01
//
//________________________________________________________________________________
//Functional description:
//
//The Binary Input Object includes the following functions
//- The input can be turned (0 = input is active) -> configuration value
//- Depending on the Parameter "in_fault_state", it is possible to select whether
//  log. 0 or log. 1 will represent the fault.
//- The input signal can be debounced in both directions with a seperate time
//  -> Real values in structure
//- The input signal can be counted -> value in structure -> configuration value
//
//The main application for the function are level indicators.
//
AUTHOR : jm
VERSION : 3.2
VAR_INPUT
  in_Handbedienung_erlaubt : BOOL ;
  in_Anlage_ein : BOOL ;
  in_Eingang : BOOL ;
  in_Eingang_drehen : BOOL ;
  in_Eingang_entprellen : BOOL ;
  in_Stoerauswertung_aktiv : BOOL ;
  in_Quitt_Stoerung_noetig : BOOL ;
  in_Stoer_Zustand : BOOL ;
  in_Quitt_Stoerung : BOOL ;
END_VAR
VAR_IN_OUT
  io_Eingang_verarbeitet : BOOL ;
  io_Stoerung : BOOL ;
  io_Struktur : ANY ;
END_VAR
VAR_TEMP
  Eingang_nach_Drehung : BOOL ;
  Eingang_nach_Entprellung : BOOL ;
  Diskrepanz : BOOL ;
  Freigabe_Entprellung_HIG : BOOL ;
  Ausgang_Entprellung_HIGH : BOOL ;
  Freigabe_Entprellung_LOW : BOOL ;
  Ausgang_Entprellung_LOW : BOOL ;
  positive_Flanke : BOOL ;
  Objektstatus : INT ;
  Temp_DB : INT ;
  Sollzeit_Entprellung_HIG : REAL ;
  Istzeit_Entprellung_HIGH : REAL ;
  Sollzeit_Entprellung_LOW : REAL ;
  Istzeit_entprellung_LOW : REAL ;
END_VAR
BEGIN
NETWORK
TITLE = Anfangs-DW der Struktur aus ANY-Zeiger auslesen
      L     P##io_Struktur;
      LAR2;
      L     D [AR2,P#6.0];
      LAR2;
NETWORK
TITLE = Daten aus Struktur lesen
      A     DIX [AR2,P#3.4];
      =     #Eingang_nach_Drehung;
      A     DIX [AR2,P#3.5];
      =     #Eingang_nach_Entprellung;
      A     DIX [AR2,P#3.6];
      =     #Ausgang_Entprellung_HIGH;
      A     DIX [AR2,P#3.7];
      =     #Ausgang_Entprellung_LOW;
      L     DID [AR2,P#8.0];
      T     #Sollzeit_Entprellung_HIG;
      L     DID [AR2,P#12.0];
      T     #Istzeit_Entprellung_HIGH;
      L     DID [AR2,P#16.0];
      T     #Sollzeit_Entprellung_LOW;
      L     DID [AR2,P#20.0];
      T     #Istzeit_entprellung_LOW;
NETWORK
TITLE = Eingang ggf. drehen
      A     #in_Eingang;
      AN    #in_Eingang_drehen;
      O;
      AN    #in_Eingang;
      A     #in_Eingang_drehen;
      =     #Eingang_nach_Drehung;
NETWORK
TITLE = Umschaltung Hand-/Automatikmode 
      A     DIX [AR2,P#2.7];	// Handmode von Farbgrafik (Struktur)
      AN    DIX [AR2,P#3.1];	// Handmode gesperrt (Struktur)
      AN    "M0.0 LockManualMode";	// Handbedienung zentral sperren 
      S     DIX [AR2,P#2.6];	// Handmode zu Farbgrafik (Struktur)
      ON    DIX [AR2,P#2.7];	// Handmode von Farbgrafik (Struktur)
      ON    #in_Handbedienung_erlaubt;
      O     "M0.0 LockManualMode";	// Handbedienung zentral sperren 
      O     DIX [AR2,P#3.1];	// Handmode gesperrt (Struktur)
      R     DIX [AR2,P#2.6];	// Handmode zu Farbgrafik (Struktur)
      R     DIX [AR2,P#2.7];	// Handmode von Farbgrafik (Struktur)
NETWORK
TITLE = Handzustand im Automatikmode speichern
      AN    DIX [AR2,P#2.6];	// Handmode zu Farbgrafik (Struktur)
      JCN   SAM;
      A     #Eingang_nach_Drehung;
      AN    #in_Eingang_drehen;
      =     DIX [AR2,P#3.0];	// Zustand Handmode (Struktur)
      AN    #Eingang_nach_Drehung;
      A     #in_Eingang_drehen;
      =     DIX [AR2,P#3.0];	// Zustand Handmode (Struktur)
SAM:  NOP   0;
NETWORK
TITLE = Zustand nach Drehung im Handmode überschreiben
      A     DIX [AR2,P#2.6];	// Handmode zu Farbgrafik (Struktur)
      JCN   SHM;
      A     DIX [AR2,P#3.0];	// Zustand Handmode (Struktur)
      =     #Eingang_nach_Drehung;
SHM:  NOP   0;
NETWORK
TITLE = Diskrepanz feststellen
// Automode
      AN    DIX [AR2,P#2.6];	// Handmode zu Farbgrafik (Struktur)
      A     #in_Stoerauswertung_aktiv;
      AN    #in_Eingang;	//Störung = log. 0
      AN    #in_Stoer_Zustand;
      O;
      AN    DIX [AR2,P#2.6];	// Handmode zu Farbgrafik (Struktur)
      A     #in_Stoerauswertung_aktiv;
      A     #in_Eingang;	//Störung = log. 1
      A     #in_Stoer_Zustand;
      O;
// Handmode 
      A     DIX [AR2,P#2.6];	// Handmode zu Farbgrafik (Struktur)
      A     #in_Stoerauswertung_aktiv;
      AN    #Eingang_nach_Drehung;	//Störung = log. 0
      AN    #in_Stoer_Zustand;
      O;
      A     DIX [AR2,P#2.6];	// Handmode zu Farbgrafik (Struktur)
      A     #in_Stoerauswertung_aktiv;
      A     #Eingang_nach_Drehung;	//Störung = log. 1
      A     #in_Stoer_Zustand;
      =     #Diskrepanz;
NETWORK
TITLE = Stoerungszaehler
      A     #in_Quitt_Stoerung_noetig;
      AN    #in_Quitt_Stoerung;
      A     #io_Stoerung;
      O;
      A     #Diskrepanz;
      AN    #in_Quitt_Stoerung;
      O;
      AN    #in_Quitt_Stoerung_noetig;
      A     #Diskrepanz;
      JC    SZ1;
      L     0;	// Wenn keine Diskrepanz dann Zähler löschen
      T     DIW [AR2,P#6.0];	// Istzeit Störung (Struktur)
      JU    ESZ;
// Störungszähler in jeder Sekunde erhöhen
SZ1:  O     #io_Stoerung;
      ON    "M4.5 ImpulseClock1,0Sec";	// Sekundenimpuls (Standardmerker)
      JC    ESZ;
      L     DIW [AR2,P#6.0];	// Istzeit Störung (Struktur)
      +     1;	// (002)
      T     DIW [AR2,P#6.0];	// Istzeit Störung (Struktur)
ESZ:  NOP   0;
NETWORK
TITLE = Störmeldung ausgeben
      L     DIW [AR2,P#6.0];	// Istzeit Störung (Struktur)
      L     DIW [AR2,P#4.0];	// Sollzeit Störung (Struktur)
      >I;
      =     #io_Stoerung;
NETWORK
TITLE = Stoerung quittieren
      O     #Diskrepanz;	// Stoerung steht noch an
      ON    #io_Stoerung;
      JC    ESQ;
      ON    #in_Quitt_Stoerung_noetig;	// Stoerung muß quittiert werden ?
      JC    SQ1;	// Stoerung muß nicht quittiert werden
      A     #in_Quitt_Stoerung;
SQ1:  R     #io_Stoerung;
ESQ:  NOP   0;
NETWORK
TITLE = Entprellung HIGH
      A     #Eingang_nach_Drehung;
      A     #in_Eingang_entprellen;
      =     #Freigabe_Entprellung_HIG;
      CALL  "FC3 Timernachbildung" (
           in_Freigabe              := #Freigabe_Entprellung_HIG,
           in_Reset                 := "M0.3 Reset",
           in_Impuls                := "M1.7 ClockTimerFunction",
           in_Impulszeit_in_100ms   := "MW 6 Timer Val Cycle FCs",
           in_Verzoegerungsart      := B#16#45,
           in_Verzoegerungszeit     := #Sollzeit_Entprellung_HIG,
           io_Ausgangssignal        := #Ausgang_Entprellung_HIGH,
           io_Zeitzaehler           := #Istzeit_Entprellung_HIGH);
NETWORK
TITLE = Entprellung LOW
      AN    #Eingang_nach_Drehung;
      A     #in_Eingang_entprellen;
      =     #Freigabe_Entprellung_LOW;
      CALL  "FC3 Timernachbildung" (
           in_Freigabe              := #Freigabe_Entprellung_LOW,
           in_Reset                 := "M0.3 Reset",
           in_Impuls                := "M1.7 ClockTimerFunction",
           in_Impulszeit_in_100ms   := "MW 6 Timer Val Cycle FCs",
           in_Verzoegerungsart      := B#16#45,
           in_Verzoegerungszeit     := #Sollzeit_Entprellung_LOW,
           io_Ausgangssignal        := #Ausgang_Entprellung_LOW,
           io_Zeitzaehler           := #Istzeit_entprellung_LOW);
NETWORK
TITLE = Entprellung
      A     #Eingang_nach_Drehung;
      A     #in_Eingang_entprellen;
      A     #Ausgang_Entprellung_HIGH;
      S     #Eingang_nach_Entprellung;
      AN    #Eingang_nach_Drehung;
      A     #in_Eingang_entprellen;
      A     #Ausgang_Entprellung_LOW;
      R     #Eingang_nach_Entprellung;
      NOP   0;
NETWORK
TITLE = verarbeitetes Eingangssignal zuweisen
// Automatikmode
      AN    DIX [AR2,P#2.6];	// Handmode zu Farbgrafik (Struktur)
      AN    #in_Eingang_entprellen;
      A     #Eingang_nach_Drehung;
//      UN    #io_Stoerung                // (006) (007)
      O;
// Automatikmode
      AN    DIX [AR2,P#2.6];	// Handmode zu Farbgrafik (Struktur)
      A     #in_Eingang_entprellen;
      A     #Eingang_nach_Entprellung;
//      UN    #io_Stoerung                // (006) (007)
      O;
// Handmode 
      A     DIX [AR2,P#2.6];	// Handmode zu Farbgrafik (Struktur)
      A     DIX [AR2,P#3.0];	// Zustand Handmode (Struktur)
      AN    #in_Eingang_drehen;
//      UN    #io_Stoerung                // (006) (007)
      O;
// Handmode 
      A     DIX [AR2,P#2.6];	// Handmode zu Farbgrafik (Struktur)
      AN    DIX [AR2,P#3.0];	// Zustand Handmode (Struktur)
      A     #in_Eingang_drehen;
//      UN    #io_Stoerung                // (006) (007)
      =     #io_Eingang_verarbeitet;
NETWORK
TITLE = Flankenauswertung Ausgang Ventil für Schalthäufigkeitzähler
      A     #io_Eingang_verarbeitet;
      FP    DIX [AR2,P#24.3];	// Flankenmerker Ausgang (Struktur)
      =     #positive_Flanke;
NETWORK
TITLE = Schalthäufigkeitzähler
      ON    DIX [AR2,P#0.3];	// Kennung Schalthäufigkeitzähler ein (Struktur)
      ON    #positive_Flanke;
      JC    ESHZ;
      L     1.000000e+00;
      L     DID [AR2,P#26.0];	// Schalthäufigkeitzähler (Struktur)
      +R;
      T     DID [AR2,P#26.0];	// Schalthäufigkeitzähler (Struktur)
ESHZ: NOP   0;
NETWORK
TITLE = Schalthäufigkeitzähler zurücksetzten
      AN    DIX [AR2,P#24.0];	// Reset Schalthäufigkeitzähler (Struktur)
      JC    E_RS;
      L     0.000000e+00;
      T     DID [AR2,P#26.0];	// Schalthäufigkeitzähler (Struktur)
      CLR;
      =     DIX [AR2,P#24.0];	// Reset Schalthäufigkeitzähler (Struktur)
E_RS: NOP   0;
NETWORK
TITLE = Warnmeldung Schalthäufigkeitszähler erzeugen
      A(;
      L     DID [AR2,P#26.0];	// Schalthäufigkeitzähler (Struktur)
      L     DID [AR2,P#30.0];	// Sollwert Warnung (Struktur)
      >R;
      );
      A(;
      L     DID [AR2,P#30.0];	// Sollwert Warnung (Struktur)
      L     0.000000e+00;
      <>R;
      );
      =     DIX [AR2,P#24.1];	// Warnmeldung Schalthäufigkeitzähler (Struktur)
NETWORK
TITLE = Alarmmeldung Schalthäufigkeitszähler erzeugen
      A(;
      L     DID [AR2,P#26.0];	// Schalthäufigkeitzähler (Struktur)
      L     DID [AR2,P#34.0];	// Sollwert Alarm (Struktur)
      >R;
      );
      A(;
      L     DID [AR2,P#34.0];	// Sollwert Alarm (Struktur)
      L     0.000000e+00;
      <>R;
      );
      =     DIX [AR2,P#24.2];	// Alarmmeldung Schalthäufigkeitzähler (Struktur)
NETWORK
TITLE =  Objektstatus für Visualisation OP (009) (010)
// 19 = Anlage nicht ein (interlock) ==> Farbvorschlag orange
      L     19;
      AN    #in_Anlage_ein;
      AN    #io_Stoerung;
      JC    disp;
// 1 = nicht betaetigt ==> Farbvorschlag weiß
      L     1;
      AN    #io_Eingang_verarbeitet;
      AN    #io_Stoerung;
      AN    DIX [AR2,P#1.0];	// Kennung "invers"
      O;
      A     #io_Eingang_verarbeitet;
      AN    #io_Stoerung;
      A     DIX [AR2,P#1.0];	// Kennung "invers"
      JC    disp;
// 5 = betätigt ==> Farbvorschlag grün(gelb)
      L     5;
      A     #io_Eingang_verarbeitet;
      AN    #io_Stoerung;
      AN    DIX [AR2,P#1.0];	// Kennung "invers"
      O;
      AN    #io_Eingang_verarbeitet;
      AN    #io_Stoerung;
      A     DIX [AR2,P#1.0];	// Kennung "invers"
      JC    disp;
// 14 = Störung, nicht betätigt, Störung ==> Farbvorschlag rot/weiß
      L     14;	// (007)
      AN    #io_Eingang_verarbeitet;	// (007)
      A     #io_Stoerung;	// (007)
      AN    DIX [AR2,P#1.0];	// (007) Kennung "invers"
      A     #in_Anlage_ein;	// (007)
      O;	// (007)
      A     #io_Eingang_verarbeitet;	// (007)
      A     #io_Stoerung;	// (007)
      A     DIX [AR2,P#1.0];	// (007) Kennung "invers"
      A     #in_Anlage_ein;	// (007)
      JC    disp;	// (007)
// 15 = Störung, nicht betätigtt, Störung ==> Farbvorschlag rot/grün(gelb)
      L     15;	// (008)
      A     #io_Eingang_verarbeitet;	// (007)
      A     #io_Stoerung;	// (007)
      AN    DIX [AR2,P#1.0];	// (007) Kennung "invers"
      A     #in_Anlage_ein;	// (007)
      O;	// (007)
      AN    #io_Eingang_verarbeitet;	// (007)
      A     #io_Stoerung;	// (007) (008)
      A     DIX [AR2,P#1.0];	// (007) Kennung "invers"
      A     #in_Anlage_ein;	// (007)
      JC    disp;	// (007)
// 16 = Störung
      L     16;
      A     #io_Stoerung;
      JC    disp;
      L     0;
disp: T     #Objektstatus;
NETWORK
TITLE = Daten in Struktur kopieren
      A     #io_Eingang_verarbeitet;
      =     DIX [AR2,P#2.0];	// Eingang verarbeitet (Struktur)
      A     #in_Eingang;
      =     DIX [AR2,P#2.1];	// Eingang (Struktur)
      A     #in_Eingang_drehen;
      =     DIX [AR2,P#2.2];	// Eingang drehen (Struktur)
      A     #in_Eingang_entprellen;
      =     DIX [AR2,P#2.3];	// Eingang entprellen (Struktur)
      A     #in_Stoer_Zustand;
      =     DIX [AR2,P#2.4];	// Störzustand (Struktur)
      A     #io_Stoerung;
      =     DIX [AR2,P#2.5];	// Störung (Struktur)
      A     #in_Anlage_ein;	// (006)
      =     DIX [AR2,P#3.2];	// (006) Anlage ein (Struktur) 
      A     #Eingang_nach_Drehung;
      =     DIX [AR2,P#3.4];
      A     #Eingang_nach_Entprellung;
      =     DIX [AR2,P#3.5];
      A     #Ausgang_Entprellung_HIGH;
      =     DIX [AR2,P#3.6];
      A     #Ausgang_Entprellung_LOW;
      =     DIX [AR2,P#3.7];
      AN    #Ausgang_Entprellung_HIGH;
      JCN   noHi;
      L     #Istzeit_Entprellung_HIGH;
      T     DID [AR2,P#12.0];
noHi: NOP   0;
      AN    #Ausgang_Entprellung_LOW;
      JCN   noLo;
      L     #Istzeit_entprellung_LOW;
      T     DID [AR2,P#20.0];
noLo: NOP   0;
      L     #Objektstatus;
      T     DIW [AR2,P#48.0];	// #Objektstatus  (Struktur) 
END_FUNCTION

FUNCTION "FC25 Lamp" : VOID	// FC 25
TITLE = Lamp Functiomnality - copied from TIA Library
NAME : standard
VERSION : 0.1
VAR_INPUT
  Steady : BOOL ;
  Flash : BOOL ;
  DoubleFlash : BOOL ;
  LampTest : BOOL ;
END_VAR
VAR_OUTPUT
  Lamp : BOOL ;
END_VAR
BEGIN
NETWORK
TITLE = Lamp Operation
      A     #Steady;
      AN    #Flash;
      AN    #DoubleFlash;
      AN    "M1.5 Lamp Test";
      O;
      A     #Flash;
      AN    #DoubleFlash;
      A     "M2.4 Flag0,8Sec";
      AN    "M1.5 Lamp Test";
      O;
      A     #DoubleFlash;
      A     "M2.4 Flag0,8Sec";
      A     "M2.1 Flag0,2Sec";
      AN    "M1.5 Lamp Test";
      O;
      A     "M1.5 Lamp Test";
      O;
      A     #LampTest;
      =     #Lamp;
END_FUNCTION

FUNCTION "AnalogueIn" : VOID	// FC 28
TITLE = Block for analog input
//Building:
//Date         Editor                                                     Version
//--------------------------------------------------------------------------------
//06.03.2017   (gea)                                                      01.00.00
//
//Modifications:
//No. Date     Edit  Description                                    Index Version
//--------------------------------------------------------------------------------
//01a 20.06.17 gea   Filter implemented                             (001) 01.01.00
//01b 17.01.18 gea   no configuration clean-up to allow dynamic     (001b)
//                   alarm enable
//________________________________________________________________________________
//Functional description:
//
//The analog Input Object includes the following functions
//- 
//
AUTHOR : gea
VERSION : 1.1
VAR_INPUT
  ManOpEn : BOOL ;	// Enable Manual mode
  ManModeTrack : BOOL ;	// Manual mode PV tracking
  OVErrEn : BOOL ;	// overflow/underflow/broken wire error enable
  AlarmHiEn : BOOL ;	// Alarm high enable
  AlarmHiAckEn : BOOL ;	// Alarm high acknowledge enable
  AlarmLoEn : BOOL ;	//Alarm low enable
  AlarmLoAckEn : BOOL ;	//Alarm low acknowledge enable
  SwitchEn : BOOL ;	//Switch enable
  SwitchPol : BOOL ;	//Switch polarity
  DigitMin : INT ;	// scaling digit max
  DigitMax : INT ;	// scaling digit min
  ValueMin : REAL ;	// scaling value max
  ValueMax : REAL ;	// scaling value min
  ValueSubs : REAL ;	// substitude value
  Filter : REAL ;	//filter value = 1.0 ...
  Configuration : WORD ;	// external Configuration (0=use internal)
  UOM : INT ;	// external Uom  (0=use internal)
  iSystemOn : BOOL ;	// System activated
  iwDigit : INT ;	// input digit value
  aAlarmHiAck : BOOL ;	// Alarm high acknowledge
  aAlarmLoAck : BOOL ;	//Alarm low acknowledge
END_VAR
VAR_IN_OUT
  PVAct : REAL ;
  Switch : BOOL ;
  fAlarmHi : BOOL ;
  fAlarmLo : BOOL ;
  fScalingErr : BOOL ;
  fOVErr : BOOL ;
  ioStructure : ANY ;
END_VAR
VAR_TEMP
  State : INT ;
  tempReal1 : REAL ;
  tempReal2 : REAL ;
  tempDB : INT ;
  PVIn : REAL ;
END_VAR
BEGIN
NETWORK
TITLE =  get start byte of structure
      L     P##ioStructure;
      LAR2;
      L     W [AR2,P#4.0];
      T     #tempDB;
      OPN   DI [#tempDB];
      L     D [AR2,P#6.0];
      LAR2;
NETWORK
TITLE =  external  configuration
      L     #Configuration;
      L     0;
      ==I;
      JC    NECO;
      L     #Configuration;
      L     0;
      <>I;
      =     DIX [AR2,P#0.0];	// AnalogInOn on
      L     #Configuration;
      L     2#1000;
      AW;
      L     0;
      <>I;
      =     DIX [AR2,P#0.3];	// switch counter on
      L     #Configuration;
      L     2#10000;
      AW;
      L     0;
      <>I;
      =     DIX [AR2,P#0.4];	// switch level input
      L     #Configuration;
      L     2#100000;
      AW;
      L     0;
      <>I;
      =     DIX [AR2,P#0.5];	// switch level hysteresis input
      L     #Configuration;
      L     2#100000000;
      AW;
      L     0;
      <>I;
      =     DIX [AR2,P#1.0];	// alarm high level input
      L     #Configuration;
      L     2#1000000000;
      AW;
      L     0;
      <>I;
      =     DIX [AR2,P#1.1];	// alarm low level input
      L     #Configuration;
      L     2#10000000000;
      AW;
      L     0;
      <>I;
      =     DIX [AR2,P#1.2];	// alarm level hysteresis input
NECO: NOP   0;
      L     #UOM;
      L     0;
      ==I;
      JC    NEUO;
      L     #UOM;
      T     DIW [AR2,P#2.0];
NEUO: NOP   0;
NETWORK
TITLE =  clean up configuration
//      UN    #SwitchEn                                                                     //(001b)
//      R     DIX [AR2,P#0.4]             // switch level input                             //(001b)
//      R     DIX [AR2,P#0.5]             // switch level hysteresis input                  //(001b)
//      R     DIX [AR2,P#0.3]             // switch counter on                              //(001b)
//      UN    #AlarmHiEn                                                                    //(001b)
//      R     DIX [AR2,P#1.0]             // alarm high level input                         //(001b)
//      UN    #AlarmLoEn                                                                    //(001b)
//      R     DIX [AR2,P#1.1]             // alarm low level input                          //(001b)
//      UN    #AlarmHiEn                                                                    //(001b)
//      UN    #AlarmLoEn                                                                    //(001b)
//      R     DIX [AR2,P#1.2]             // alarm level hysteresis input                   //(001b)
NETWORK
TITLE =  selection manual mode
      A     DIX [AR2,P#4.1];	// ManModeOp
      AN    DIX [AR2,P#4.2];	// ManModeLock
      AN    "M0.0 LockManualMode";	// manual mode general disabled
      S     DIX [AR2,P#4.0];	// ManModAct
      ON    DIX [AR2,P#4.1];	// ManModeOp
      ON    #ManOpEn;	// manual mode local disabled
      O     "M0.0 LockManualMode";	// manual mode general disabled
      O     DIX [AR2,P#4.2];	// ManModeLock
      R     DIX [AR2,P#4.0];	// ManModAct
      R     DIX [AR2,P#4.1];	// ManModeOp
NETWORK
TITLE =  overflow / underflow / broken wire check
      O(;
      L     #iwDigit;
      L     32511;
      >I;
      );	//overflow
      O(;
      A(;
      L     #iwDigit;
      L     -32512;
      <I;
      );
      A(;
      L     #DigitMin;
      L     0;
      <>I;	//bipolar
      );
      );	//underflow bipolar
      O(;
      A(;
      L     #iwDigit;
      L     -4864;
      <I;
      );
      A(;
      L     #DigitMin;
      L     0;
      ==I;	//unipolar
      );
      );	//underflow //unipolar
      A     #OVErrEn;	//enable overflow / underflow error
      =     #fOVErr;
NETWORK
TITLE =  scaling of PV
//Val = ValueMin + (ValueMax-ValueMin)*(iwDigit-DigitMin)/(DigitMax-DigitMin)
// (network holds code this reader does not know; not shown)
NETWORK
TITLE =  substidue PV
      O     #fScalingErr;
      O     #fOVErr;
      AN    DIX [AR2,P#4.0];	// ManModAct
      JCN   PVSU;
      L     #ValueSubs;
      T     #PVIn;	//(001)
PVSU: NOP   0;
NETWORK
TITLE = manual mode PV
      A     DIX [AR2,P#4.0];	// ManModAct
      JCN   PVMA;
      L     DID [AR2,P#10.0];	//ManModePV      
      T     #PVIn;	//(001)
PVMA: NOP   0;
NETWORK
TITLE = Filter PV
//(001) 
// 
      L     1.000000e+00;
      L     #Filter;
      <R;
      JC    FIOK;
      L     #PVIn;	//in case the number of counts is 0 or negative
      JU    FNOK;
FIOK: L     1.000000e+00;
      -R;
      L     #PVAct;
      *R;
      L     #PVIn;
      +R;
      L     #Filter;
      /R;
FNOK: T     #PVAct;
NETWORK
TITLE =  track manual mode value in automatic
      AN    DIX [AR2,P#4.0];	// ManModAct
      A     #ManModeTrack;
      JCN   PVTK;
      L     #PVAct;
      T     DID [AR2,P#10.0];	//ManModePV      
PVTK: NOP   0;
NETWORK
TITLE = Alarm high
      A(;
      L     #PVAct;
      L     DID [AR2,P#14.0];	//AlarmHiPV
      >R;	//PVact>AlarmHiPV
      );
      A     #AlarmHiEn;
      S     #fAlarmHi;
      A(;
      L     DID [AR2,P#14.0];	//AlarmHiPV
      L     DID [AR2,P#22.0];	//AlarmHystPV
      -R;
      L     #PVAct;
      TAK;
      <R;	//PVact<(AlarmHiPV-AlarmHystPV
      );
      A(;
      A     #AlarmHiAckEn;
      A     #aAlarmHiAck;
      ON    #AlarmHiAckEn;
      );
      ON    #AlarmHiEn;
      ON    #iSystemOn;
      R     #fAlarmHi;
NETWORK
TITLE = Alarm low
      A(;
      L     #PVAct;
      L     DID [AR2,P#18.0];	//AlarmLoPV
      <R;	//PVact<AlarmLoPV
      );
      A     #AlarmLoEn;
      S     #fAlarmLo;
      A(;
      L     DID [AR2,P#18.0];	//AlarmLoPV
      L     DID [AR2,P#22.0];	//AlarmHystPV
      +R;
      L     #PVAct;
      TAK;
      >R;	//PVact<(AlarmHiPV-AlarmHystPV
      );
      A(;
      A     #AlarmLoAckEn;
      A     #aAlarmLoAck;
      ON    #AlarmLoAckEn;
      );
      ON    #AlarmLoEn;
      ON    #iSystemOn;
      R     #fAlarmLo;
NETWORK
TITLE = switch
      L     DID [AR2,P#26.0];	//SwitchLevelPV
      L     DID [AR2,P#30.0];	//SwitchHysteresis
      -R;
      T     #tempReal1;	//Switch level high hysteresis
      L     DID [AR2,P#26.0];	//SwitchLevelPV
      L     DID [AR2,P#30.0];	//SwitchHysteresis
      +R;
      T     #tempReal2;	//Switch level low hysteresis
      A     #SwitchEn;
      A     #SwitchPol;
      A(;
      L     #PVAct;
      L     DID [AR2,P#26.0];	//SwitchLevelPV
      >R;
      );	//(SwitchPolarity=positive) * (PVAct>SwitchLevel)
      O;
      A     #SwitchEn;
      AN    #SwitchPol;
      A(;
      L     #PVAct;
      L     DID [AR2,P#26.0];	//SwitchLevelPV
      <R;
      );	//(SwitchPolarity=negative) * (PVAct<SwitchLevel)
      S     #Switch;
      A     #SwitchEn;
      A     #SwitchPol;
      A(;
      L     #PVAct;
      L     #tempReal1;	//Switch level high hysteresis
      <R;
      );	//(SwitchPolarity=positive) * (PVAct<(SwitchLevel-SwitchLevelhysteresis)
      O;
      A     #SwitchEn;
      AN    #SwitchPol;
      A(;
      L     #PVAct;
      L     #tempReal2;	//Switch level low hysteresis
      >R;
      );	//(SwitchPolarity=negative) * (PVAct<(SwitchLevel+SwitchLevelhysteresis)
      ON    #SwitchEn;
      R     #Switch;
NETWORK
TITLE =  Switch counter count up
      A     #Switch;
      FP    DIX [AR2,P#34.3];	// Switch counter edge
      A     DIX [AR2,P#0.3];	// Configuarion switching counter
      JCN   SCUP;
      L     1.000000e+00;
      L     DID [AR2,P#36.0];	// Switch counter
      +R;
      T     DID [AR2,P#36.0];	// Switch counter
SCUP: NOP   0;
NETWORK
TITLE =  Switch counter reset
      A     DIX [AR2,P#34.0];	// Switch counter Reset
      JCN   SCRE;
      R     DIX [AR2,P#34.0];	// Switch counter Reset
      L     0.000000e+00;
      T     DID [AR2,P#36.0];	// Switch counter
SCRE: NOP   0;
NETWORK
TITLE = Switch counter warning
      A(;
      L     DID [AR2,P#36.0];	// Switch counter
      L     DID [AR2,P#40.0];	// Switch counter warning count
      >R;
      );
      A(;
      L     DID [AR2,P#40.0];	// Switch counter warning count
      L     0.000000e+00;
      <>R;
      );
      =     DIX [AR2,P#34.1];	// Switch counter warning 
NETWORK
TITLE = Switch counter alarm
      A(;
      L     DID [AR2,P#36.0];	// Switch counter
      L     DID [AR2,P#44.0];	// Switch counter alarm count
      >R;
      );
      A(;
      L     DID [AR2,P#44.0];	// Sollwert Alarm (Struktur)
      L     0.000000e+00;
      <>R;
      );
      =     DIX [AR2,P#34.2];	// Switch counter alarm 
NETWORK
TITLE =  Objektstatus für Visualisation OP (009) (010)
// 9 = scaling/overflow/underflow/broken wire: substitude value ==> grey 
      L     9;
      O     #fScalingErr;
      O     #fOVErr;
      JC    disp;
// 19 = system not on (interlock) ==> orange
      L     19;
      AN    #iSystemOn;
      JC    disp;
// 16 = alarm high ==> red
      L     16;
      O     #fAlarmHi;
      JC    disp;
// 16 = alarm low ==> yellow
      L     13;
      O     #fAlarmLo;
      JC    disp;
// 5 = switch on ==> green
      L     5;
      A     #Switch;
      A     #SwitchEn;
      JC    disp;
// 1 = switch off ==> white
      L     1;
      AN    #Switch;
      A     #SwitchEn;
      JC    disp;
      L     0;
disp: T     #State;
NETWORK
TITLE =  save data to structure
      A     #iSystemOn;
      =     DIX [AR2,P#4.3];
      A     #fScalingErr;
      =     DIX [AR2,P#4.4];
      A     #fOVErr;
      =     DIX [AR2,P#4.5];
      A     #fAlarmHi;
      =     DIX [AR2,P#4.6];
      A     #AlarmHiEn;
      =     DIX [AR2,P#4.7];
      A     #aAlarmHiAck;
      =     DIX [AR2,P#5.0];
      A     #fAlarmLo;
      =     DIX [AR2,P#5.1];
      A     #AlarmLoEn;
      =     DIX [AR2,P#5.2];
      A     #aAlarmLoAck;
      =     DIX [AR2,P#5.3];
      L     #PVAct;
      T     DID [AR2,P#6.0];
      A     #Switch;
      =     DIX [AR2,P#5.4];
      A     #SwitchEn;
      =     DIX [AR2,P#5.5];
      L     #State;
      T     DIW [AR2,P#48.0];	// #Objektstatus  (Struktur) 
END_FUNCTION

